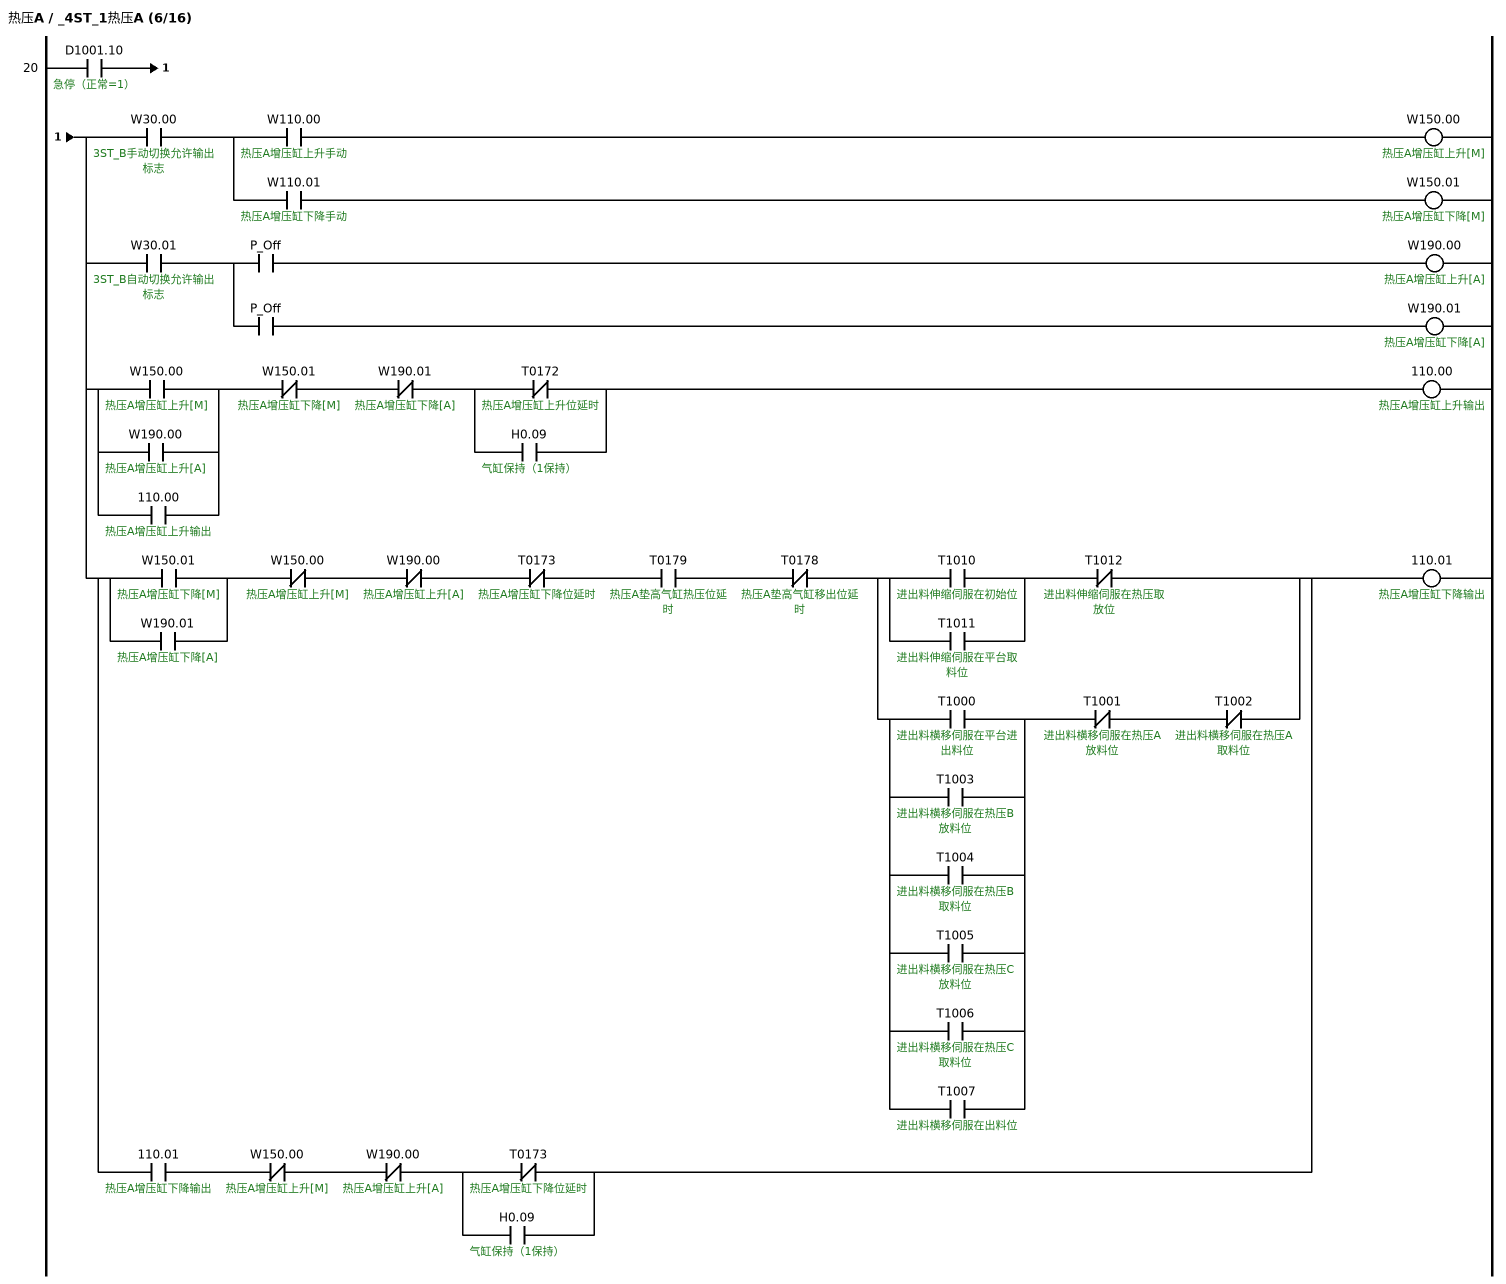
; [picture p144: 热压A / _4ST_1热压A, rungs 20-20]
; rung 20
LD D1001.10  ; 急停（正常=1）
OUT TR0
AND W30.00  ; 3ST_B手动切换允许输出标志
OUT TR1
AND W110.00  ; 热压A增压缸上升手动
OUT W150.00  ; 热压A增压缸上升[M]
LD TR1
AND W110.01  ; 热压A增压缸下降手动
OUT W150.01  ; 热压A增压缸下降[M]
LD TR0
AND W30.01  ; 3ST_B自动切换允许输出标志
OUT TR1
AND P_Off
OUT W190.00  ; 热压A增压缸上升[A]
LD TR1
AND P_Off
OUT W190.01  ; 热压A增压缸下降[A]
LD TR0
LD W150.00  ; 热压A增压缸上升[M]
OR W190.00  ; 热压A增压缸上升[A]
OR 110.00  ; 热压A增压缸上升输出
ANDLD
ANDNOT W150.01  ; 热压A增压缸下降[M]
ANDNOT W190.01  ; 热压A增压缸下降[A]
LDNOT T0172  ; 热压A增压缸上升位延时
OR H0.09  ; 气缸保持（1保持）
ANDLD
OUT 110.00  ; 热压A增压缸上升输出
LD TR0
LD W150.01  ; 热压A增压缸下降[M]
OR W190.01  ; 热压A增压缸下降[A]
ANDNOT W150.00  ; 热压A增压缸上升[M]
ANDNOT W190.00  ; 热压A增压缸上升[A]
ANDNOT T0173  ; 热压A增压缸下降位延时
AND T0179  ; 热压A垫高气缸热压位延时
ANDNOT T0178  ; 热压A垫高气缸移出位延时
LD T1010  ; 进出料伸缩伺服在初始位
OR T1011  ; 进出料伸缩伺服在平台取料位
ANDNOT T1012  ; 进出料伸缩伺服在热压取放位
LD T1000  ; 进出料横移伺服在平台进出料位
OR T1003  ; 进出料横移伺服在热压B放料位
OR T1004  ; 进出料横移伺服在热压B取料位
OR T1005  ; 进出料横移伺服在热压C放料位
OR T1006  ; 进出料横移伺服在热压C取料位
OR T1007  ; 进出料横移伺服在出料位
ANDNOT T1001  ; 进出料横移伺服在热压A放料位
ANDNOT T1002  ; 进出料横移伺服在热压A取料位
ORLD
ANDLD
LD 110.01  ; 热压A增压缸下降输出
ANDNOT W150.00  ; 热压A增压缸上升[M]
ANDNOT W190.00  ; 热压A增压缸上升[A]
LDNOT T0173  ; 热压A增压缸下降位延时
OR H0.09  ; 气缸保持（1保持）
ANDLD
ORLD
ANDLD
OUT 110.01  ; 热压A增压缸下降输出

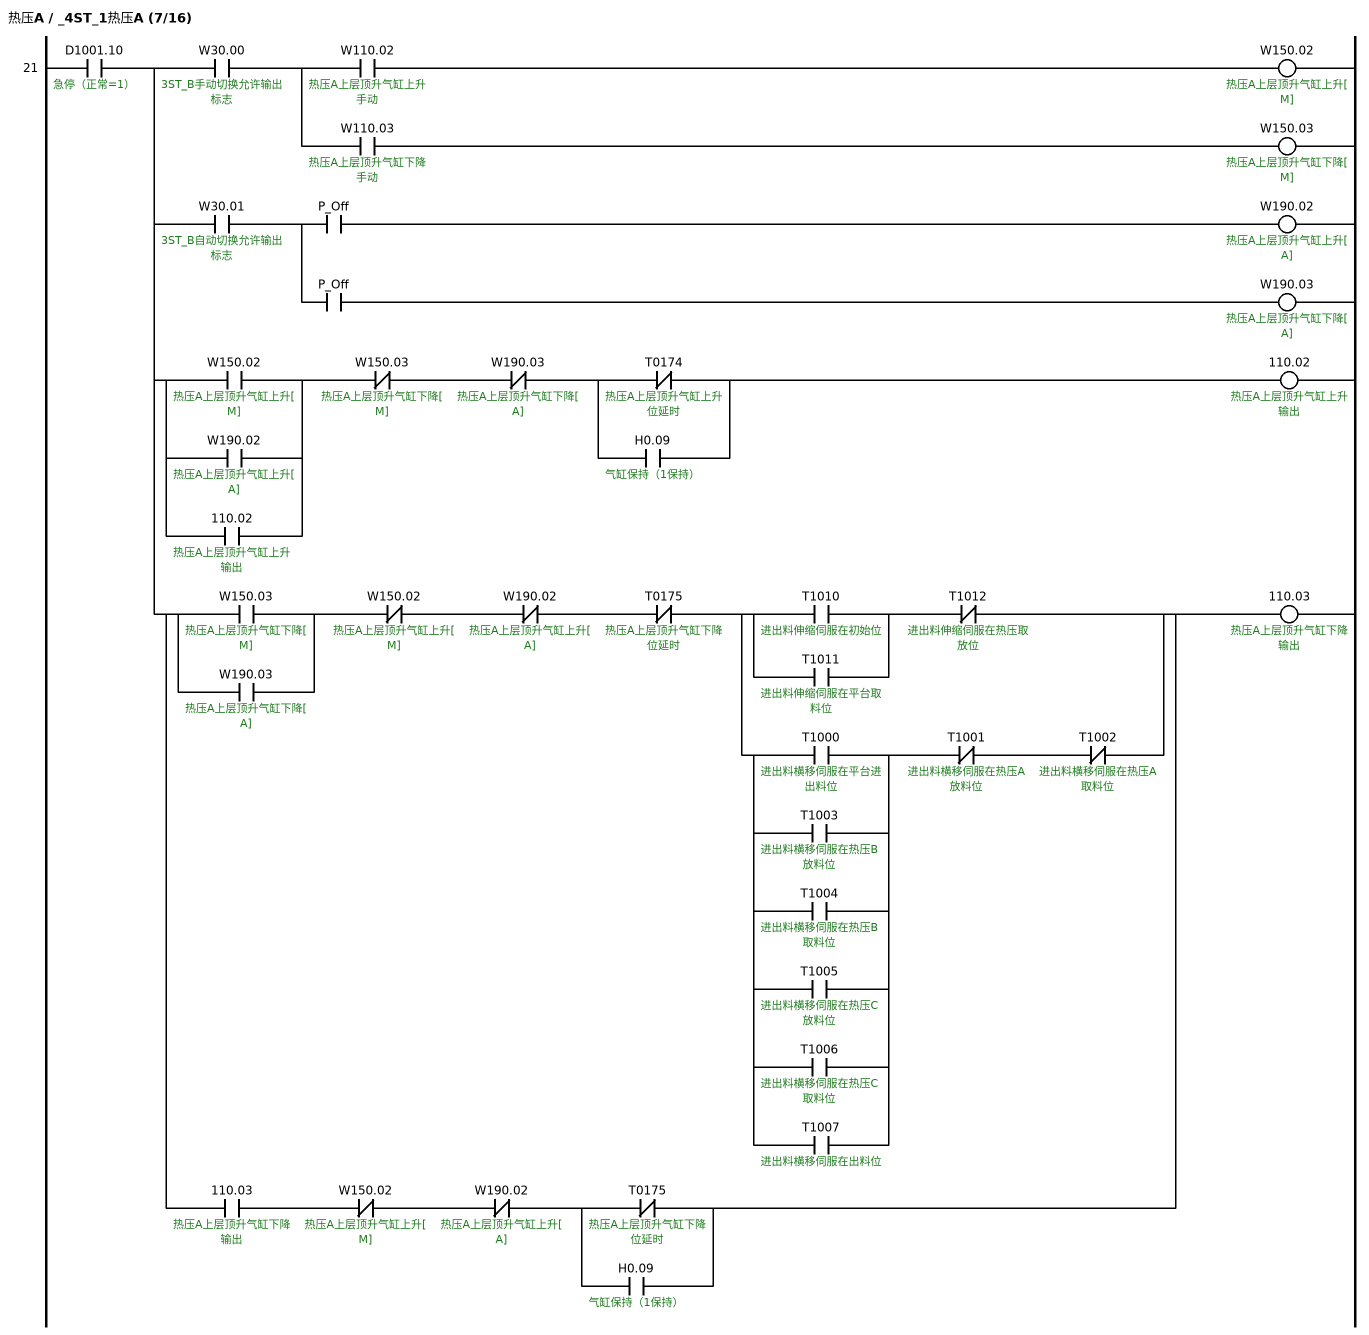
; rung 21
LD D1001.10  ; 急停（正常=1）
OUT TR0
AND W30.00  ; 3ST_B手动切换允许输出标志
OUT TR1
AND W110.02  ; 热压A上层顶升气缸上升手动
OUT W150.02  ; 热压A上层顶升气缸上升[M]
LD TR1
AND W110.03  ; 热压A上层顶升气缸下降手动
OUT W150.03  ; 热压A上层顶升气缸下降[M]
LD TR0
AND W30.01  ; 3ST_B自动切换允许输出标志
OUT TR1
AND P_Off
OUT W190.02  ; 热压A上层顶升气缸上升[A]
LD TR1
AND P_Off
OUT W190.03  ; 热压A上层顶升气缸下降[A]
LD TR0
LD W150.02  ; 热压A上层顶升气缸上升[M]
OR W190.02  ; 热压A上层顶升气缸上升[A]
OR 110.02  ; 热压A上层顶升气缸上升输出
ANDLD
ANDNOT W150.03  ; 热压A上层顶升气缸下降[M]
ANDNOT W190.03  ; 热压A上层顶升气缸下降[A]
LDNOT T0174  ; 热压A上层顶升气缸上升位延时
OR H0.09  ; 气缸保持（1保持）
ANDLD
OUT 110.02  ; 热压A上层顶升气缸上升输出
LD TR0
LD W150.03  ; 热压A上层顶升气缸下降[M]
OR W190.03  ; 热压A上层顶升气缸下降[A]
ANDNOT W150.02  ; 热压A上层顶升气缸上升[M]
ANDNOT W190.02  ; 热压A上层顶升气缸上升[A]
ANDNOT T0175  ; 热压A上层顶升气缸下降位延时
LD T1010  ; 进出料伸缩伺服在初始位
OR T1011  ; 进出料伸缩伺服在平台取料位
ANDNOT T1012  ; 进出料伸缩伺服在热压取放位
LD T1000  ; 进出料横移伺服在平台进出料位
OR T1003  ; 进出料横移伺服在热压B放料位
OR T1004  ; 进出料横移伺服在热压B取料位
OR T1005  ; 进出料横移伺服在热压C放料位
OR T1006  ; 进出料横移伺服在热压C取料位
OR T1007  ; 进出料横移伺服在出料位
ANDNOT T1001  ; 进出料横移伺服在热压A放料位
ANDNOT T1002  ; 进出料横移伺服在热压A取料位
ORLD
ANDLD
LD 110.03  ; 热压A上层顶升气缸下降输出
ANDNOT W150.02  ; 热压A上层顶升气缸上升[M]
ANDNOT W190.02  ; 热压A上层顶升气缸上升[A]
LDNOT T0175  ; 热压A上层顶升气缸下降位延时
OR H0.09  ; 气缸保持（1保持）
ANDLD
ORLD
ANDLD
OUT 110.03  ; 热压A上层顶升气缸下降输出

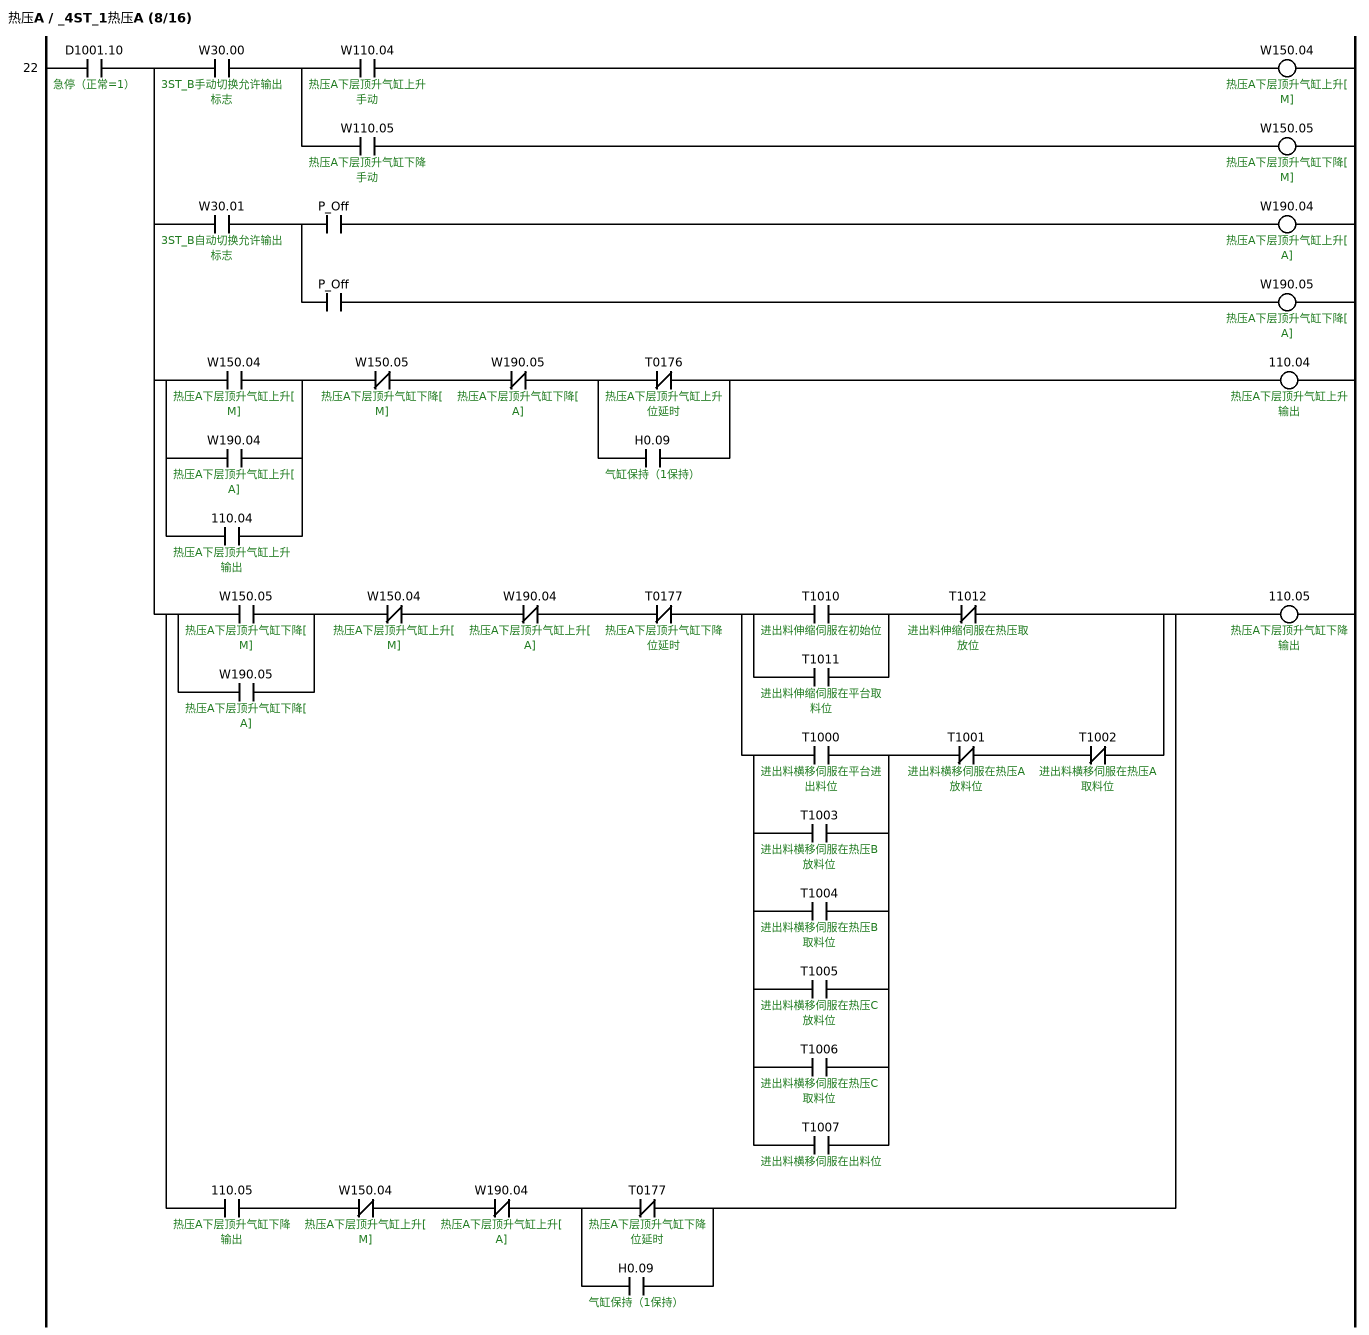
; rung 22
LD D1001.10  ; 急停（正常=1）
OUT TR0
AND W30.00  ; 3ST_B手动切换允许输出标志
OUT TR1
AND W110.04  ; 热压A下层顶升气缸上升手动
OUT W150.04  ; 热压A下层顶升气缸上升[M]
LD TR1
AND W110.05  ; 热压A下层顶升气缸下降手动
OUT W150.05  ; 热压A下层顶升气缸下降[M]
LD TR0
AND W30.01  ; 3ST_B自动切换允许输出标志
OUT TR1
AND P_Off
OUT W190.04  ; 热压A下层顶升气缸上升[A]
LD TR1
AND P_Off
OUT W190.05  ; 热压A下层顶升气缸下降[A]
LD TR0
LD W150.04  ; 热压A下层顶升气缸上升[M]
OR W190.04  ; 热压A下层顶升气缸上升[A]
OR 110.04  ; 热压A下层顶升气缸上升输出
ANDLD
ANDNOT W150.05  ; 热压A下层顶升气缸下降[M]
ANDNOT W190.05  ; 热压A下层顶升气缸下降[A]
LDNOT T0176  ; 热压A下层顶升气缸上升位延时
OR H0.09  ; 气缸保持（1保持）
ANDLD
OUT 110.04  ; 热压A下层顶升气缸上升输出
LD TR0
LD W150.05  ; 热压A下层顶升气缸下降[M]
OR W190.05  ; 热压A下层顶升气缸下降[A]
ANDNOT W150.04  ; 热压A下层顶升气缸上升[M]
ANDNOT W190.04  ; 热压A下层顶升气缸上升[A]
ANDNOT T0177  ; 热压A下层顶升气缸下降位延时
LD T1010  ; 进出料伸缩伺服在初始位
OR T1011  ; 进出料伸缩伺服在平台取料位
ANDNOT T1012  ; 进出料伸缩伺服在热压取放位
LD T1000  ; 进出料横移伺服在平台进出料位
OR T1003  ; 进出料横移伺服在热压B放料位
OR T1004  ; 进出料横移伺服在热压B取料位
OR T1005  ; 进出料横移伺服在热压C放料位
OR T1006  ; 进出料横移伺服在热压C取料位
OR T1007  ; 进出料横移伺服在出料位
ANDNOT T1001  ; 进出料横移伺服在热压A放料位
ANDNOT T1002  ; 进出料横移伺服在热压A取料位
ORLD
ANDLD
LD 110.05  ; 热压A下层顶升气缸下降输出
ANDNOT W150.04  ; 热压A下层顶升气缸上升[M]
ANDNOT W190.04  ; 热压A下层顶升气缸上升[A]
LDNOT T0177  ; 热压A下层顶升气缸下降位延时
OR H0.09  ; 气缸保持（1保持）
ANDLD
ORLD
ANDLD
OUT 110.05  ; 热压A下层顶升气缸下降输出

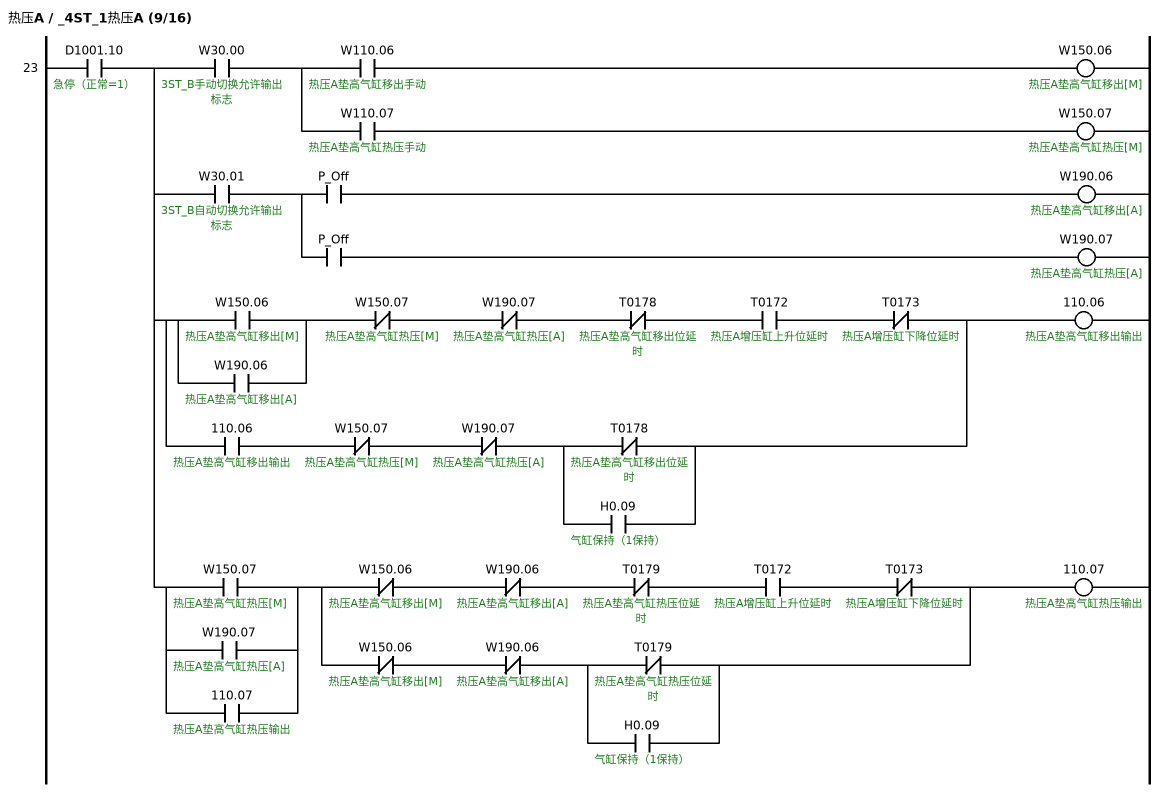
; rung 23
LD D1001.10  ; 急停（正常=1）
OUT TR0
AND W30.00  ; 3ST_B手动切换允许输出标志
OUT TR1
AND W110.06  ; 热压A垫高气缸移出手动
OUT W150.06  ; 热压A垫高气缸移出[M]
LD TR1
AND W110.07  ; 热压A垫高气缸热压手动
OUT W150.07  ; 热压A垫高气缸热压[M]
LD TR0
AND W30.01  ; 3ST_B自动切换允许输出标志
OUT TR1
AND P_Off
OUT W190.06  ; 热压A垫高气缸移出[A]
LD TR1
AND P_Off
OUT W190.07  ; 热压A垫高气缸热压[A]
LD TR0
LD W150.06  ; 热压A垫高气缸移出[M]
OR W190.06  ; 热压A垫高气缸移出[A]
ANDNOT W150.07  ; 热压A垫高气缸热压[M]
ANDNOT W190.07  ; 热压A垫高气缸热压[A]
ANDNOT T0178  ; 热压A垫高气缸移出位延时
AND T0172  ; 热压A增压缸上升位延时
ANDNOT T0173  ; 热压A增压缸下降位延时
LD 110.06  ; 热压A垫高气缸移出输出
ANDNOT W150.07  ; 热压A垫高气缸热压[M]
ANDNOT W190.07  ; 热压A垫高气缸热压[A]
LDNOT T0178  ; 热压A垫高气缸移出位延时
OR H0.09  ; 气缸保持（1保持）
ANDLD
ORLD
ANDLD
OUT 110.06  ; 热压A垫高气缸移出输出
LD TR0
LD W150.07  ; 热压A垫高气缸热压[M]
OR W190.07  ; 热压A垫高气缸热压[A]
OR 110.07  ; 热压A垫高气缸热压输出
ANDLD
LDNOT W150.06  ; 热压A垫高气缸移出[M]
ANDNOT W190.06  ; 热压A垫高气缸移出[A]
ANDNOT T0179  ; 热压A垫高气缸热压位延时
AND T0172  ; 热压A增压缸上升位延时
ANDNOT T0173  ; 热压A增压缸下降位延时
LDNOT W150.06  ; 热压A垫高气缸移出[M]
ANDNOT W190.06  ; 热压A垫高气缸移出[A]
LDNOT T0179  ; 热压A垫高气缸热压位延时
OR H0.09  ; 气缸保持（1保持）
ANDLD
ORLD
ANDLD
OUT 110.07  ; 热压A垫高气缸热压输出

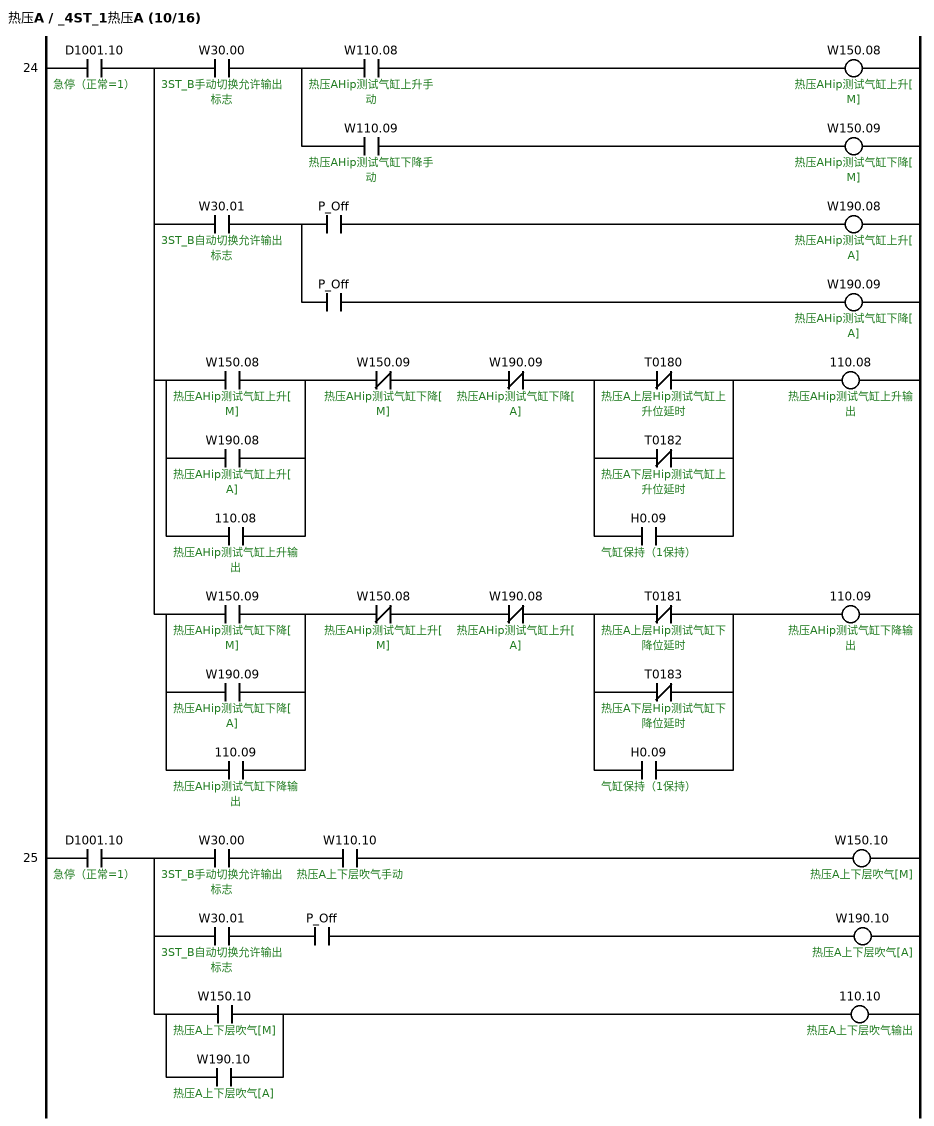
; rung 24
LD D1001.10  ; 急停（正常=1）
OUT TR0
AND W30.00  ; 3ST_B手动切换允许输出标志
OUT TR1
AND W110.08  ; 热压AHip测试气缸上升手动
OUT W150.08  ; 热压AHip测试气缸上升[M]
LD TR1
AND W110.09  ; 热压AHip测试气缸下降手动
OUT W150.09  ; 热压AHip测试气缸下降[M]
LD TR0
AND W30.01  ; 3ST_B自动切换允许输出标志
OUT TR1
AND P_Off
OUT W190.08  ; 热压AHip测试气缸上升[A]
LD TR1
AND P_Off
OUT W190.09  ; 热压AHip测试气缸下降[A]
LD TR0
LD W150.08  ; 热压AHip测试气缸上升[M]
OR W190.08  ; 热压AHip测试气缸上升[A]
OR 110.08  ; 热压AHip测试气缸上升输出
ANDLD
ANDNOT W150.09  ; 热压AHip测试气缸下降[M]
ANDNOT W190.09  ; 热压AHip测试气缸下降[A]
LDNOT T0180  ; 热压A上层Hip测试气缸上升位延时
ORNOT T0182  ; 热压A下层Hip测试气缸上升位延时
OR H0.09  ; 气缸保持（1保持）
ANDLD
OUT 110.08  ; 热压AHip测试气缸上升输出
LD TR0
LD W150.09  ; 热压AHip测试气缸下降[M]
OR W190.09  ; 热压AHip测试气缸下降[A]
OR 110.09  ; 热压AHip测试气缸下降输出
ANDLD
ANDNOT W150.08  ; 热压AHip测试气缸上升[M]
ANDNOT W190.08  ; 热压AHip测试气缸上升[A]
LDNOT T0181  ; 热压A上层Hip测试气缸下降位延时
ORNOT T0183  ; 热压A下层Hip测试气缸下降位延时
OR H0.09  ; 气缸保持（1保持）
ANDLD
OUT 110.09  ; 热压AHip测试气缸下降输出
; rung 25
LD D1001.10  ; 急停（正常=1）
OUT TR0
AND W30.00  ; 3ST_B手动切换允许输出标志
AND W110.10  ; 热压A上下层吹气手动
OUT W150.10  ; 热压A上下层吹气[M]
LD TR0
AND W30.01  ; 3ST_B自动切换允许输出标志
AND P_Off
OUT W190.10  ; 热压A上下层吹气[A]
LD TR0
LD W150.10  ; 热压A上下层吹气[M]
OR W190.10  ; 热压A上下层吹气[A]
ANDLD
OUT 110.10  ; 热压A上下层吹气输出

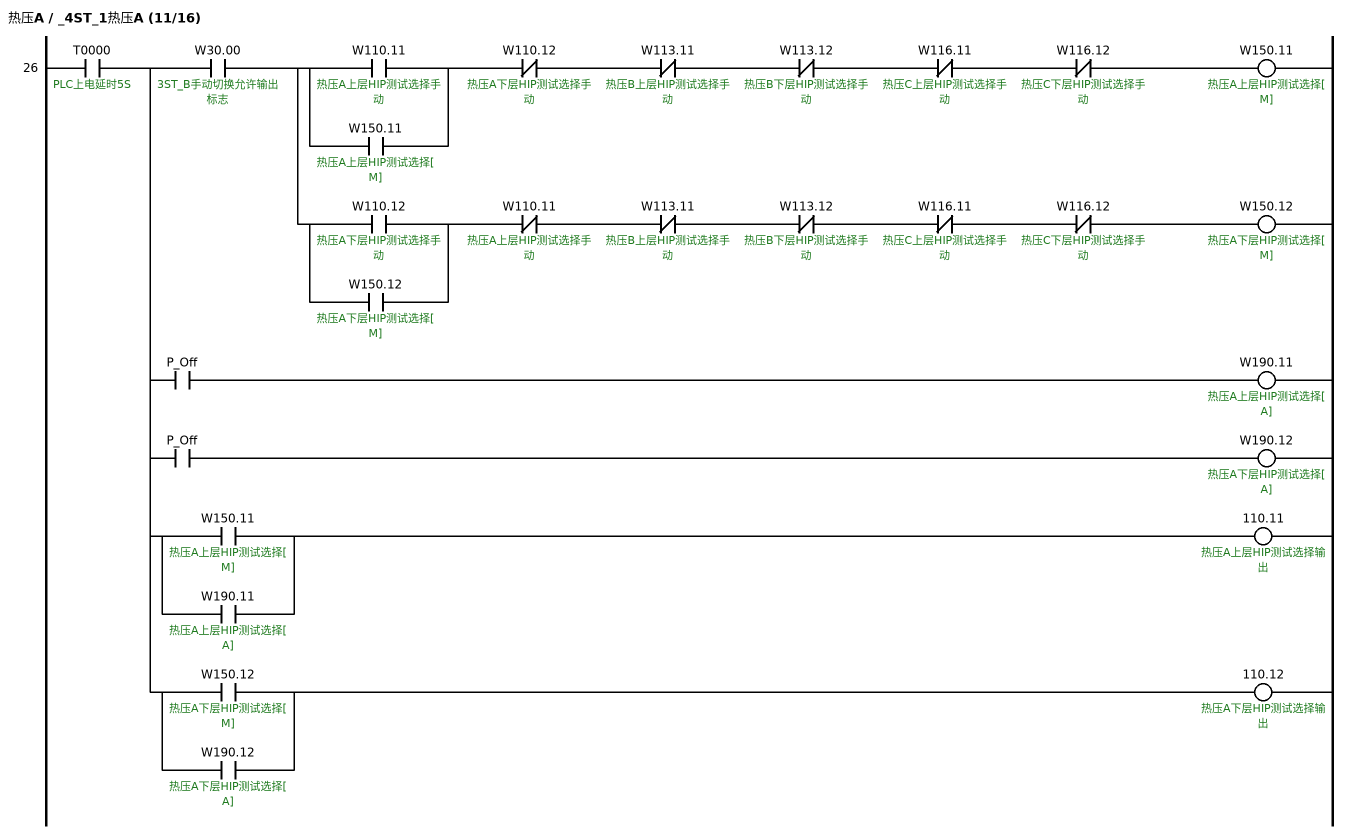
; rung 26
LD T0000  ; PLC上电延时5S
OUT TR0
AND W30.00  ; 3ST_B手动切换允许输出标志
OUT TR1
LD W110.11  ; 热压A上层HIP测试选择手动
OR W150.11  ; 热压A上层HIP测试选择[M]
ANDLD
ANDNOT W110.12  ; 热压A下层HIP测试选择手动
ANDNOT W113.11  ; 热压B上层HIP测试选择手动
ANDNOT W113.12  ; 热压B下层HIP测试选择手动
ANDNOT W116.11  ; 热压C上层HIP测试选择手动
ANDNOT W116.12  ; 热压C下层HIP测试选择手动
OUT W150.11  ; 热压A上层HIP测试选择[M]
LD TR1
LD W110.12  ; 热压A下层HIP测试选择手动
OR W150.12  ; 热压A下层HIP测试选择[M]
ANDLD
ANDNOT W110.11  ; 热压A上层HIP测试选择手动
ANDNOT W113.11  ; 热压B上层HIP测试选择手动
ANDNOT W113.12  ; 热压B下层HIP测试选择手动
ANDNOT W116.11  ; 热压C上层HIP测试选择手动
ANDNOT W116.12  ; 热压C下层HIP测试选择手动
OUT W150.12  ; 热压A下层HIP测试选择[M]
LD TR0
AND P_Off
OUT W190.11  ; 热压A上层HIP测试选择[A]
LD TR0
AND P_Off
OUT W190.12  ; 热压A下层HIP测试选择[A]
LD TR0
LD W150.11  ; 热压A上层HIP测试选择[M]
OR W190.11  ; 热压A上层HIP测试选择[A]
ANDLD
OUT 110.11  ; 热压A上层HIP测试选择输出
LD TR0
LD W150.12  ; 热压A下层HIP测试选择[M]
OR W190.12  ; 热压A下层HIP测试选择[A]
ANDLD
OUT 110.12  ; 热压A下层HIP测试选择输出

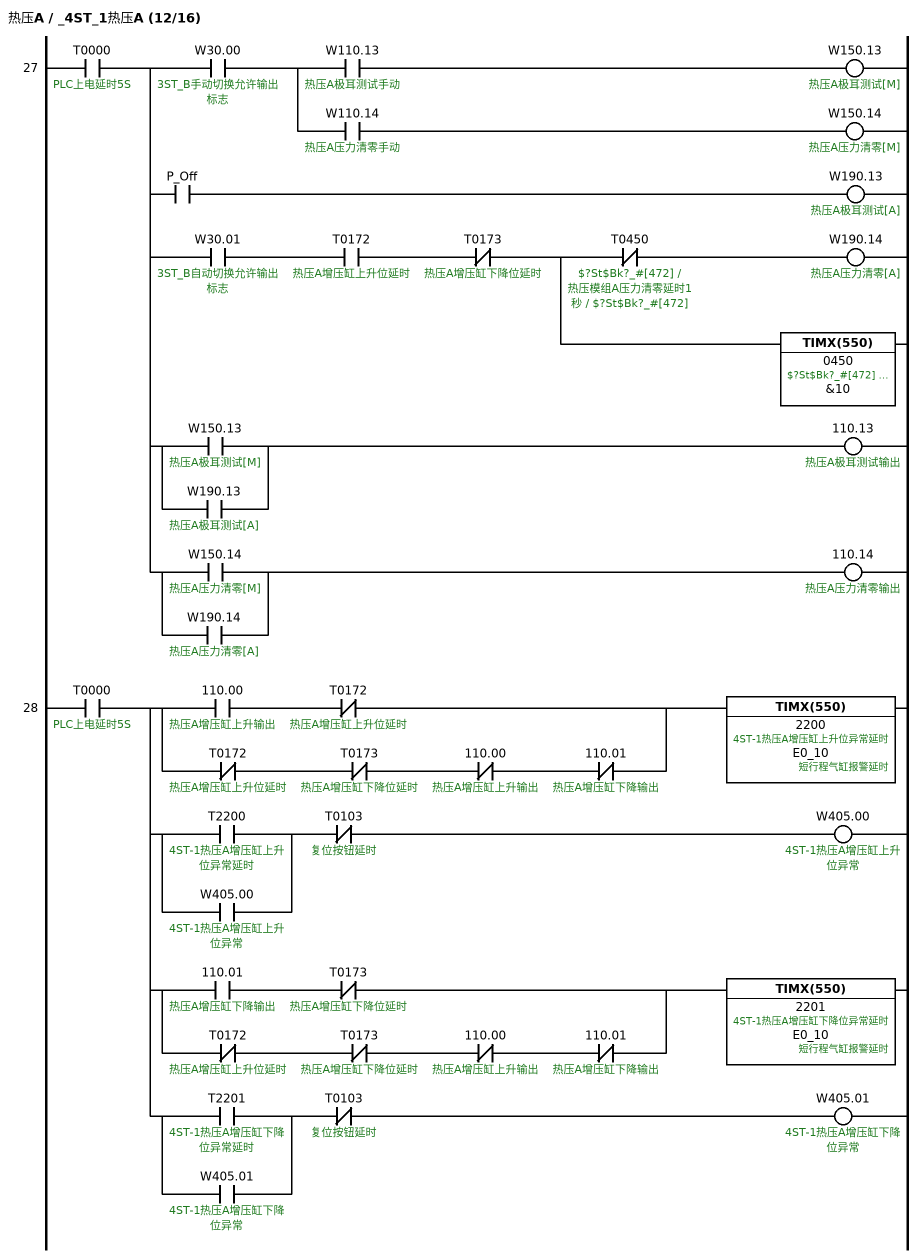
; rung 27
LD T0000  ; PLC上电延时5S
OUT TR0
AND W30.00  ; 3ST_B手动切换允许输出标志
OUT TR1
AND W110.13  ; 热压A极耳测试手动
OUT W150.13  ; 热压A极耳测试[M]
LD TR1
AND W110.14  ; 热压A压力清零手动
OUT W150.14  ; 热压A压力清零[M]
LD TR0
AND P_Off
OUT W190.13  ; 热压A极耳测试[A]
LD TR0
AND W30.01  ; 3ST_B自动切换允许输出标志
AND T0172  ; 热压A增压缸上升位延时
ANDNOT T0173  ; 热压A增压缸下降位延时
OUT TR1
ANDNOT T0450  ; $?St$Bk?_#[472] / 热压模组A压力清零延时1秒 / $?St$Bk?_#[472]
OUT W190.14  ; 热压A压力清零[A]
LD TR1
TIMX(550) 0450 &10  ; $?St$Bk?_#[472] / 热压模组A压力清零延时1秒 / $?St$Bk?_#[472]
LD TR0
LD W150.13  ; 热压A极耳测试[M]
OR W190.13  ; 热压A极耳测试[A]
ANDLD
OUT 110.13  ; 热压A极耳测试输出
LD TR0
LD W150.14  ; 热压A压力清零[M]
OR W190.14  ; 热压A压力清零[A]
ANDLD
OUT 110.14  ; 热压A压力清零输出
; rung 28
LD T0000  ; PLC上电延时5S
OUT TR0
LD 110.00  ; 热压A增压缸上升输出
ANDNOT T0172  ; 热压A增压缸上升位延时
LDNOT T0172  ; 热压A增压缸上升位延时
ANDNOT T0173  ; 热压A增压缸下降位延时
ANDNOT 110.00  ; 热压A增压缸上升输出
ANDNOT 110.01  ; 热压A增压缸下降输出
ORLD
ANDLD
TIMX(550) 2200 E0_10  ; 短行程气缸报警延时, 4ST-1热压A增压缸上升位异常延时
LD TR0
LD T2200  ; 4ST-1热压A增压缸上升位异常延时
OR W405.00  ; 4ST-1热压A增压缸上升位异常
ANDLD
ANDNOT T0103  ; 复位按钮延时
OUT W405.00  ; 4ST-1热压A增压缸上升位异常
LD TR0
LD 110.01  ; 热压A增压缸下降输出
ANDNOT T0173  ; 热压A增压缸下降位延时
LDNOT T0172  ; 热压A增压缸上升位延时
ANDNOT T0173  ; 热压A增压缸下降位延时
ANDNOT 110.00  ; 热压A增压缸上升输出
ANDNOT 110.01  ; 热压A增压缸下降输出
ORLD
ANDLD
TIMX(550) 2201 E0_10  ; 短行程气缸报警延时, 4ST-1热压A增压缸下降位异常延时
LD TR0
LD T2201  ; 4ST-1热压A增压缸下降位异常延时
OR W405.01  ; 4ST-1热压A增压缸下降位异常
ANDLD
ANDNOT T0103  ; 复位按钮延时
OUT W405.01  ; 4ST-1热压A增压缸下降位异常

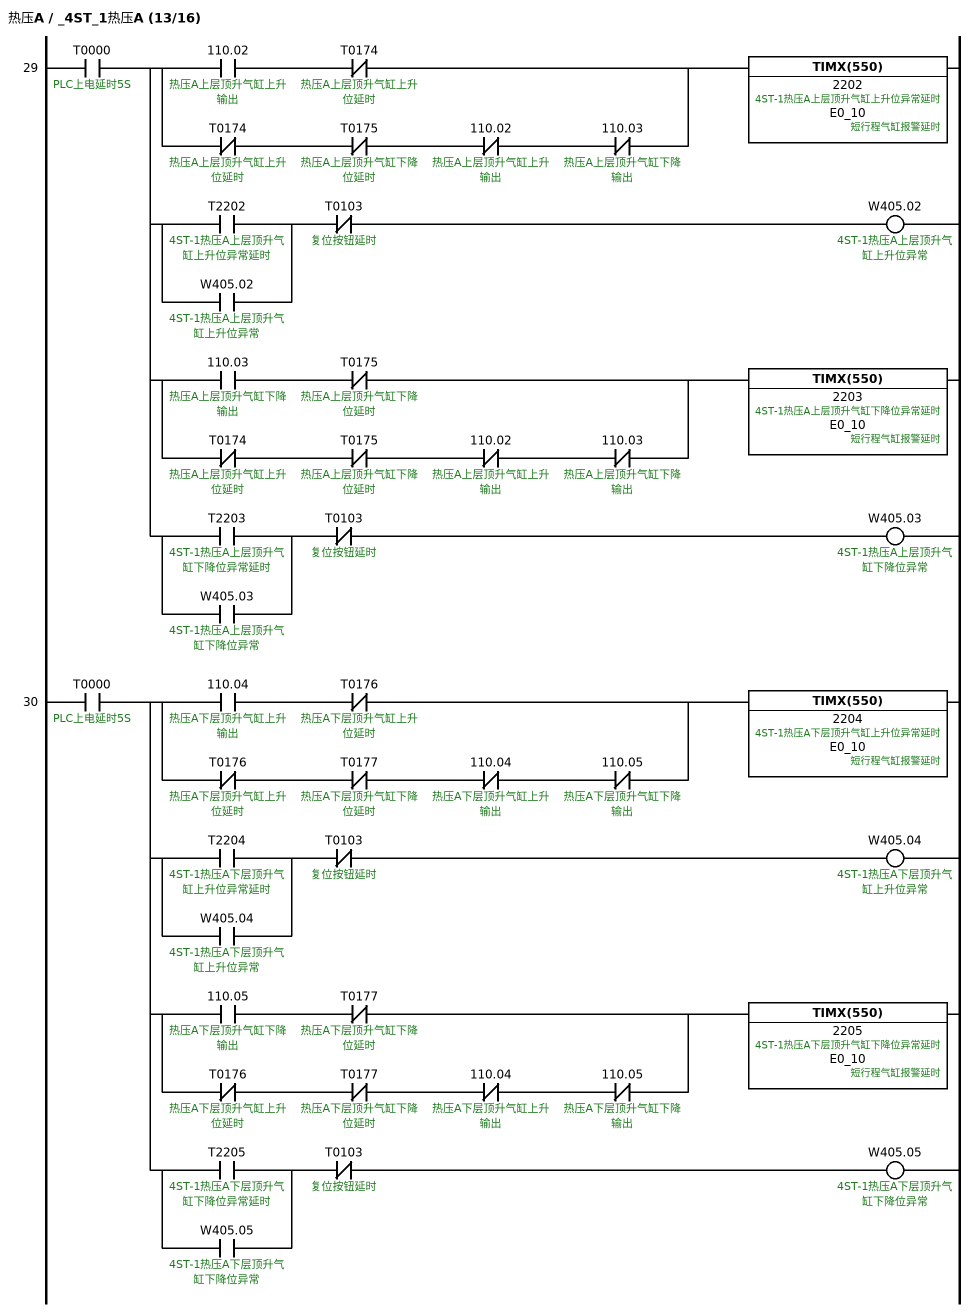
; rung 29
LD T0000  ; PLC上电延时5S
OUT TR0
LD 110.02  ; 热压A上层顶升气缸上升输出
ANDNOT T0174  ; 热压A上层顶升气缸上升位延时
LDNOT T0174  ; 热压A上层顶升气缸上升位延时
ANDNOT T0175  ; 热压A上层顶升气缸下降位延时
ANDNOT 110.02  ; 热压A上层顶升气缸上升输出
ANDNOT 110.03  ; 热压A上层顶升气缸下降输出
ORLD
ANDLD
TIMX(550) 2202 E0_10  ; 短行程气缸报警延时, 4ST-1热压A上层顶升气缸上升位异常延时
LD TR0
LD T2202  ; 4ST-1热压A上层顶升气缸上升位异常延时
OR W405.02  ; 4ST-1热压A上层顶升气缸上升位异常
ANDLD
ANDNOT T0103  ; 复位按钮延时
OUT W405.02  ; 4ST-1热压A上层顶升气缸上升位异常
LD TR0
LD 110.03  ; 热压A上层顶升气缸下降输出
ANDNOT T0175  ; 热压A上层顶升气缸下降位延时
LDNOT T0174  ; 热压A上层顶升气缸上升位延时
ANDNOT T0175  ; 热压A上层顶升气缸下降位延时
ANDNOT 110.02  ; 热压A上层顶升气缸上升输出
ANDNOT 110.03  ; 热压A上层顶升气缸下降输出
ORLD
ANDLD
TIMX(550) 2203 E0_10  ; 短行程气缸报警延时, 4ST-1热压A上层顶升气缸下降位异常延时
LD TR0
LD T2203  ; 4ST-1热压A上层顶升气缸下降位异常延时
OR W405.03  ; 4ST-1热压A上层顶升气缸下降位异常
ANDLD
ANDNOT T0103  ; 复位按钮延时
OUT W405.03  ; 4ST-1热压A上层顶升气缸下降位异常
; rung 30
LD T0000  ; PLC上电延时5S
OUT TR0
LD 110.04  ; 热压A下层顶升气缸上升输出
ANDNOT T0176  ; 热压A下层顶升气缸上升位延时
LDNOT T0176  ; 热压A下层顶升气缸上升位延时
ANDNOT T0177  ; 热压A下层顶升气缸下降位延时
ANDNOT 110.04  ; 热压A下层顶升气缸上升输出
ANDNOT 110.05  ; 热压A下层顶升气缸下降输出
ORLD
ANDLD
TIMX(550) 2204 E0_10  ; 短行程气缸报警延时, 4ST-1热压A下层顶升气缸上升位异常延时
LD TR0
LD T2204  ; 4ST-1热压A下层顶升气缸上升位异常延时
OR W405.04  ; 4ST-1热压A下层顶升气缸上升位异常
ANDLD
ANDNOT T0103  ; 复位按钮延时
OUT W405.04  ; 4ST-1热压A下层顶升气缸上升位异常
LD TR0
LD 110.05  ; 热压A下层顶升气缸下降输出
ANDNOT T0177  ; 热压A下层顶升气缸下降位延时
LDNOT T0176  ; 热压A下层顶升气缸上升位延时
ANDNOT T0177  ; 热压A下层顶升气缸下降位延时
ANDNOT 110.04  ; 热压A下层顶升气缸上升输出
ANDNOT 110.05  ; 热压A下层顶升气缸下降输出
ORLD
ANDLD
TIMX(550) 2205 E0_10  ; 短行程气缸报警延时, 4ST-1热压A下层顶升气缸下降位异常延时
LD TR0
LD T2205  ; 4ST-1热压A下层顶升气缸下降位异常延时
OR W405.05  ; 4ST-1热压A下层顶升气缸下降位异常
ANDLD
ANDNOT T0103  ; 复位按钮延时
OUT W405.05  ; 4ST-1热压A下层顶升气缸下降位异常

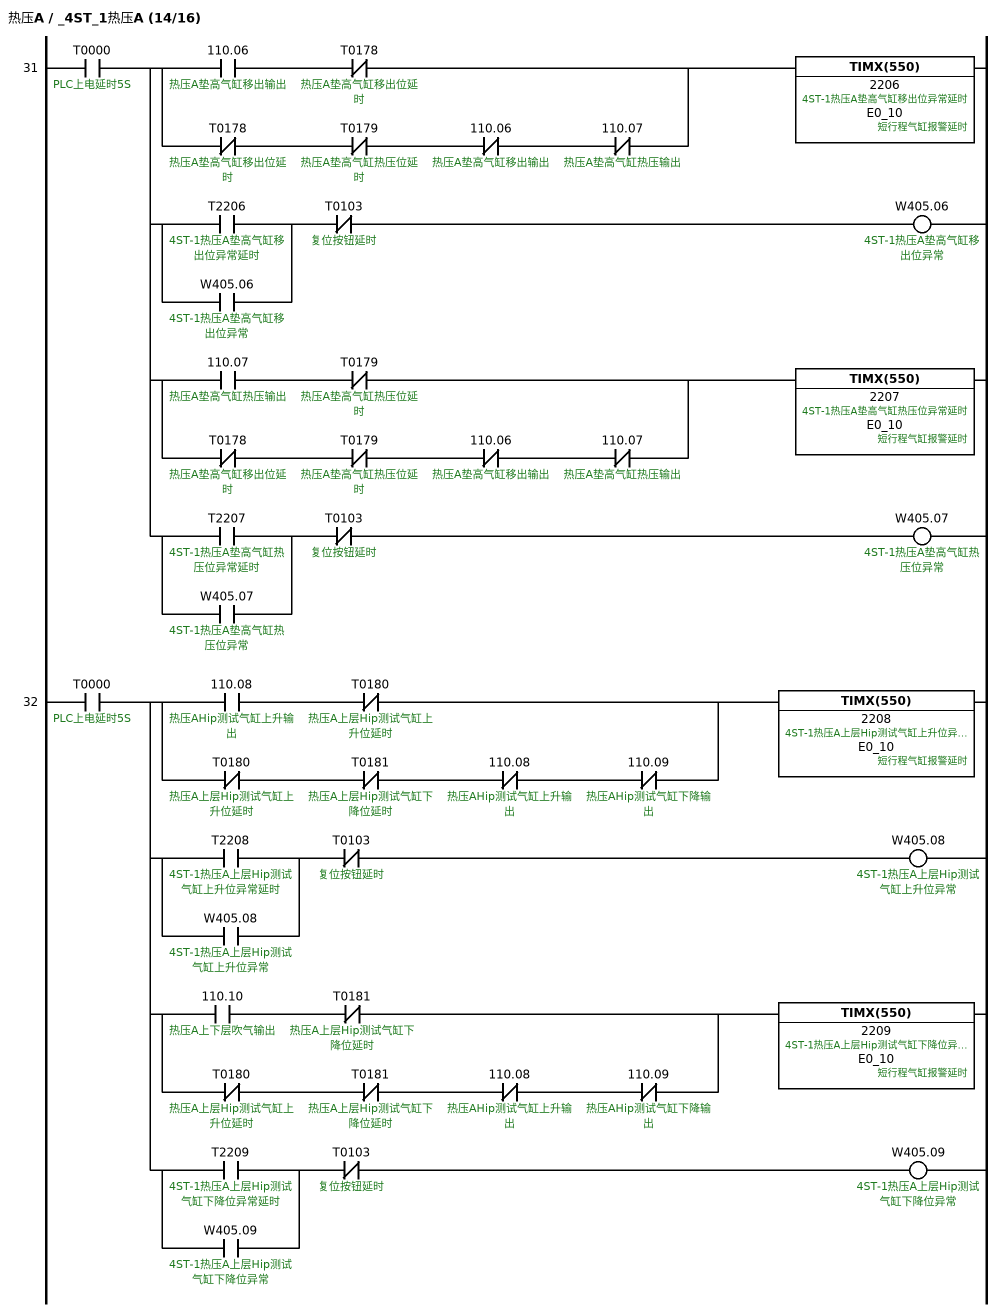
; rung 31
LD T0000  ; PLC上电延时5S
OUT TR0
LD 110.06  ; 热压A垫高气缸移出输出
ANDNOT T0178  ; 热压A垫高气缸移出位延时
LDNOT T0178  ; 热压A垫高气缸移出位延时
ANDNOT T0179  ; 热压A垫高气缸热压位延时
ANDNOT 110.06  ; 热压A垫高气缸移出输出
ANDNOT 110.07  ; 热压A垫高气缸热压输出
ORLD
ANDLD
TIMX(550) 2206 E0_10  ; 短行程气缸报警延时, 4ST-1热压A垫高气缸移出位异常延时
LD TR0
LD T2206  ; 4ST-1热压A垫高气缸移出位异常延时
OR W405.06  ; 4ST-1热压A垫高气缸移出位异常
ANDLD
ANDNOT T0103  ; 复位按钮延时
OUT W405.06  ; 4ST-1热压A垫高气缸移出位异常
LD TR0
LD 110.07  ; 热压A垫高气缸热压输出
ANDNOT T0179  ; 热压A垫高气缸热压位延时
LDNOT T0178  ; 热压A垫高气缸移出位延时
ANDNOT T0179  ; 热压A垫高气缸热压位延时
ANDNOT 110.06  ; 热压A垫高气缸移出输出
ANDNOT 110.07  ; 热压A垫高气缸热压输出
ORLD
ANDLD
TIMX(550) 2207 E0_10  ; 短行程气缸报警延时, 4ST-1热压A垫高气缸热压位异常延时
LD TR0
LD T2207  ; 4ST-1热压A垫高气缸热压位异常延时
OR W405.07  ; 4ST-1热压A垫高气缸热压位异常
ANDLD
ANDNOT T0103  ; 复位按钮延时
OUT W405.07  ; 4ST-1热压A垫高气缸热压位异常
; rung 32
LD T0000  ; PLC上电延时5S
OUT TR0
LD 110.08  ; 热压AHip测试气缸上升输出
ANDNOT T0180  ; 热压A上层Hip测试气缸上升位延时
LDNOT T0180  ; 热压A上层Hip测试气缸上升位延时
ANDNOT T0181  ; 热压A上层Hip测试气缸下降位延时
ANDNOT 110.08  ; 热压AHip测试气缸上升输出
ANDNOT 110.09  ; 热压AHip测试气缸下降输出
ORLD
ANDLD
TIMX(550) 2208 E0_10  ; 短行程气缸报警延时, 4ST-1热压A上层Hip测试气缸上升位异常延时
LD TR0
LD T2208  ; 4ST-1热压A上层Hip测试气缸上升位异常延时
OR W405.08  ; 4ST-1热压A上层Hip测试气缸上升位异常
ANDLD
ANDNOT T0103  ; 复位按钮延时
OUT W405.08  ; 4ST-1热压A上层Hip测试气缸上升位异常
LD TR0
LD 110.10  ; 热压A上下层吹气输出
ANDNOT T0181  ; 热压A上层Hip测试气缸下降位延时
LDNOT T0180  ; 热压A上层Hip测试气缸上升位延时
ANDNOT T0181  ; 热压A上层Hip测试气缸下降位延时
ANDNOT 110.08  ; 热压AHip测试气缸上升输出
ANDNOT 110.09  ; 热压AHip测试气缸下降输出
ORLD
ANDLD
TIMX(550) 2209 E0_10  ; 短行程气缸报警延时, 4ST-1热压A上层Hip测试气缸下降位异常延时
LD TR0
LD T2209  ; 4ST-1热压A上层Hip测试气缸下降位异常延时
OR W405.09  ; 4ST-1热压A上层Hip测试气缸下降位异常
ANDLD
ANDNOT T0103  ; 复位按钮延时
OUT W405.09  ; 4ST-1热压A上层Hip测试气缸下降位异常

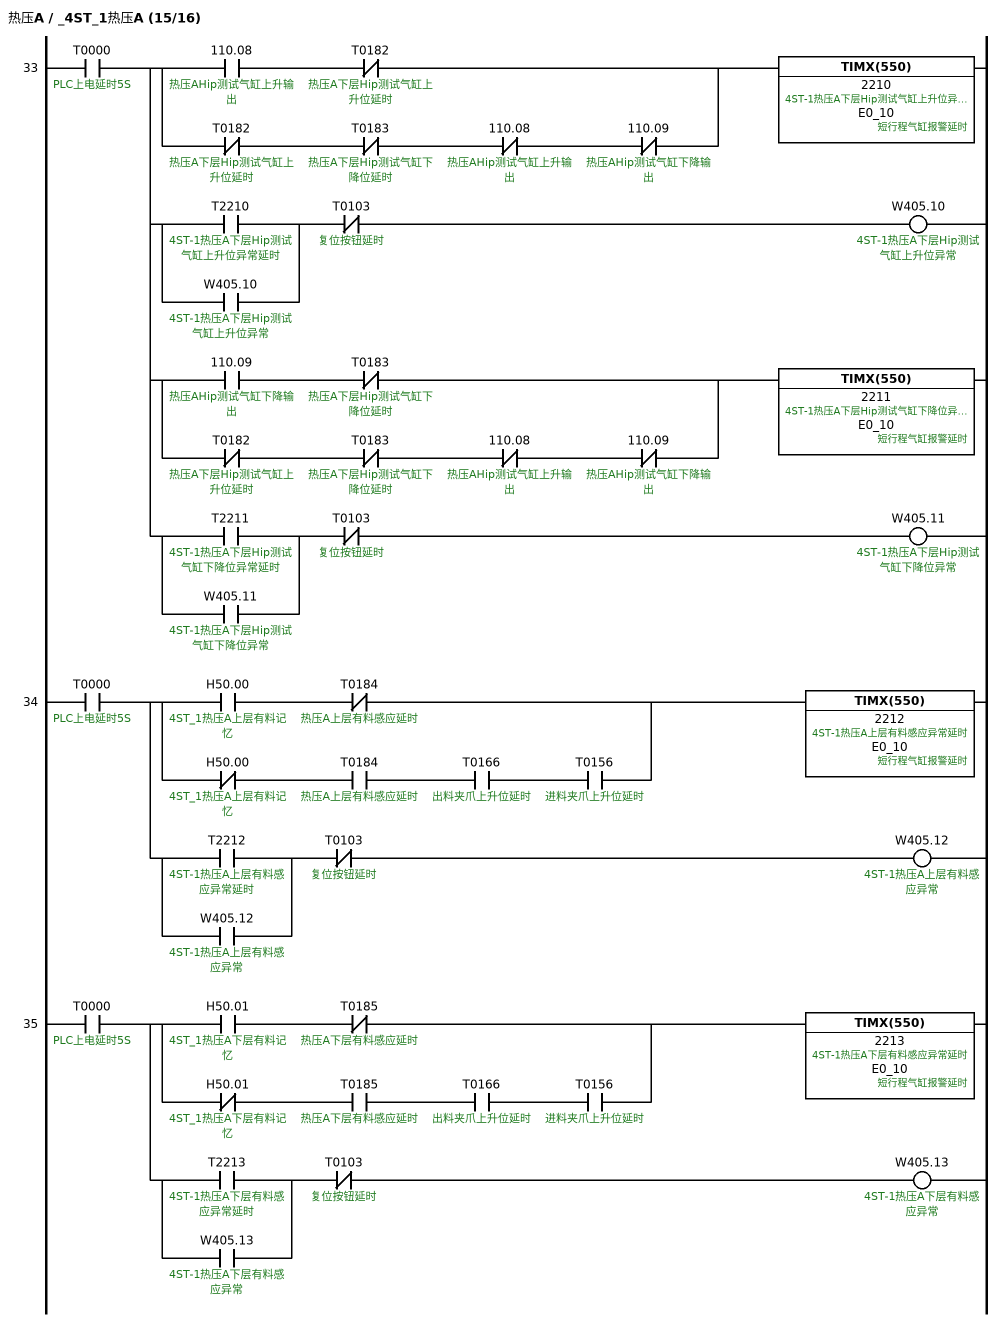
; rung 33
LD T0000  ; PLC上电延时5S
OUT TR0
LD 110.08  ; 热压AHip测试气缸上升输出
ANDNOT T0182  ; 热压A下层Hip测试气缸上升位延时
LDNOT T0182  ; 热压A下层Hip测试气缸上升位延时
ANDNOT T0183  ; 热压A下层Hip测试气缸下降位延时
ANDNOT 110.08  ; 热压AHip测试气缸上升输出
ANDNOT 110.09  ; 热压AHip测试气缸下降输出
ORLD
ANDLD
TIMX(550) 2210 E0_10  ; 短行程气缸报警延时, 4ST-1热压A下层Hip测试气缸上升位异常延时
LD TR0
LD T2210  ; 4ST-1热压A下层Hip测试气缸上升位异常延时
OR W405.10  ; 4ST-1热压A下层Hip测试气缸上升位异常
ANDLD
ANDNOT T0103  ; 复位按钮延时
OUT W405.10  ; 4ST-1热压A下层Hip测试气缸上升位异常
LD TR0
LD 110.09  ; 热压AHip测试气缸下降输出
ANDNOT T0183  ; 热压A下层Hip测试气缸下降位延时
LDNOT T0182  ; 热压A下层Hip测试气缸上升位延时
ANDNOT T0183  ; 热压A下层Hip测试气缸下降位延时
ANDNOT 110.08  ; 热压AHip测试气缸上升输出
ANDNOT 110.09  ; 热压AHip测试气缸下降输出
ORLD
ANDLD
TIMX(550) 2211 E0_10  ; 短行程气缸报警延时, 4ST-1热压A下层Hip测试气缸下降位异常延时
LD TR0
LD T2211  ; 4ST-1热压A下层Hip测试气缸下降位异常延时
OR W405.11  ; 4ST-1热压A下层Hip测试气缸下降位异常
ANDLD
ANDNOT T0103  ; 复位按钮延时
OUT W405.11  ; 4ST-1热压A下层Hip测试气缸下降位异常
; rung 34
LD T0000  ; PLC上电延时5S
OUT TR0
LD H50.00  ; 4ST_1热压A上层有料记忆
ANDNOT T0184  ; 热压A上层有料感应延时
LDNOT H50.00  ; 4ST_1热压A上层有料记忆
AND T0184  ; 热压A上层有料感应延时
AND T0166  ; 出料夹爪上升位延时
AND T0156  ; 进料夹爪上升位延时
ORLD
ANDLD
TIMX(550) 2212 E0_10  ; 短行程气缸报警延时, 4ST-1热压A上层有料感应异常延时
LD TR0
LD T2212  ; 4ST-1热压A上层有料感应异常延时
OR W405.12  ; 4ST-1热压A上层有料感应异常
ANDLD
ANDNOT T0103  ; 复位按钮延时
OUT W405.12  ; 4ST-1热压A上层有料感应异常
; rung 35
LD T0000  ; PLC上电延时5S
OUT TR0
LD H50.01  ; 4ST_1热压A下层有料记忆
ANDNOT T0185  ; 热压A下层有料感应延时
LDNOT H50.01  ; 4ST_1热压A下层有料记忆
AND T0185  ; 热压A下层有料感应延时
AND T0166  ; 出料夹爪上升位延时
AND T0156  ; 进料夹爪上升位延时
ORLD
ANDLD
TIMX(550) 2213 E0_10  ; 短行程气缸报警延时, 4ST-1热压A下层有料感应异常延时
LD TR0
LD T2213  ; 4ST-1热压A下层有料感应异常延时
OR W405.13  ; 4ST-1热压A下层有料感应异常
ANDLD
ANDNOT T0103  ; 复位按钮延时
OUT W405.13  ; 4ST-1热压A下层有料感应异常

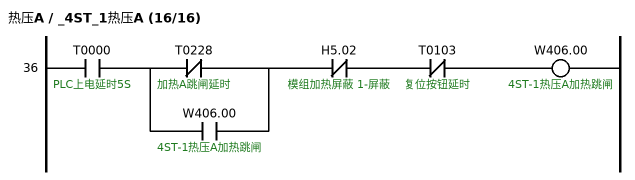
; rung 36
LD T0000  ; PLC上电延时5S
LDNOT T0228  ; 加热A跳闸延时
OR W406.00  ; 4ST-1热压A加热跳闸
ANDLD
ANDNOT H5.02  ; 模组加热屏蔽 1-屏蔽
ANDNOT T0103  ; 复位按钮延时
OUT W406.00  ; 4ST-1热压A加热跳闸

### Section 复位

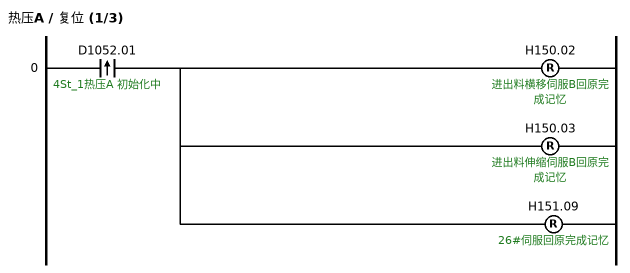
; rung 0
@LD D1052.01  ; 4St_1热压A 初始化中
RSET H150.02  ; 进出料横移伺服B回原完成记忆
RSET H150.03  ; 进出料伸缩伺服B回原完成记忆
RSET H151.09  ; 26#伺服回原完成记忆

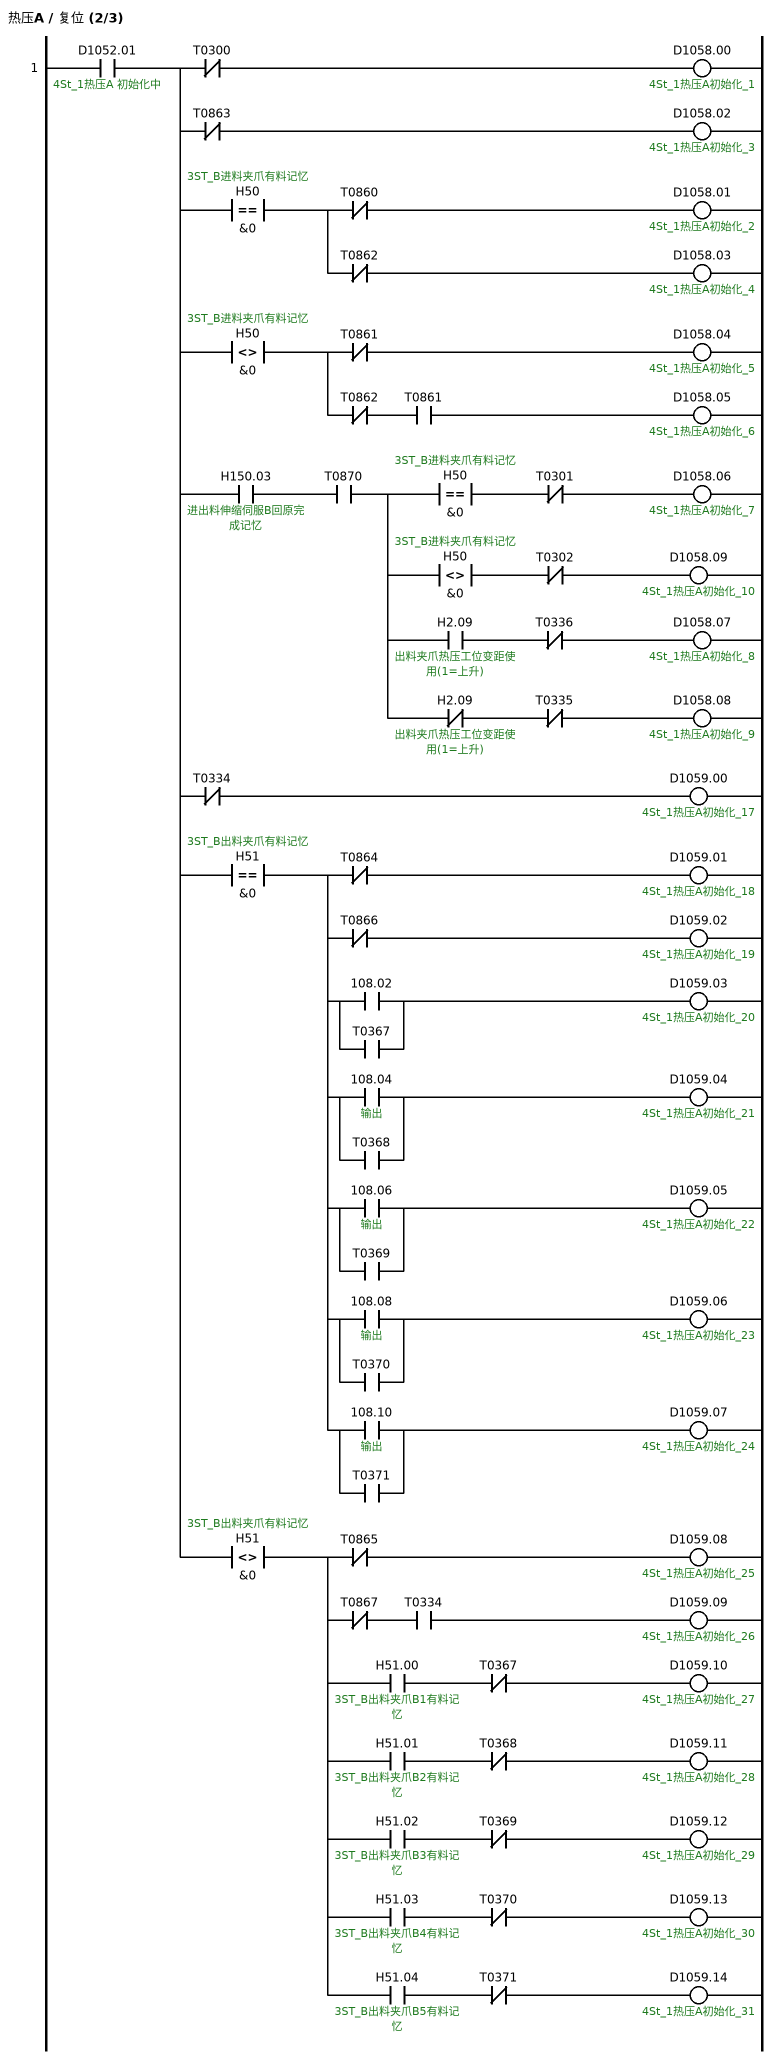
; rung 1
LD D1052.01  ; 4St_1热压A 初始化中
OUT TR0
ANDNOT T0300
OUT D1058.00  ; 4St_1热压A初始化_1
LD TR0
ANDNOT T0863
OUT D1058.02  ; 4St_1热压A初始化_3
LD TR0
AND=(300) H50 &0  ; 3ST_B进料夹爪有料记忆
OUT TR1
ANDNOT T0860
OUT D1058.01  ; 4St_1热压A初始化_2
LD TR1
ANDNOT T0862
OUT D1058.03  ; 4St_1热压A初始化_4
LD TR0
AND<>(305) H50 &0  ; 3ST_B进料夹爪有料记忆
OUT TR1
ANDNOT T0861
OUT D1058.04  ; 4St_1热压A初始化_5
LD TR1
ANDNOT T0862
AND T0861
OUT D1058.05  ; 4St_1热压A初始化_6
LD TR0
AND H150.03  ; 进出料伸缩伺服B回原完成记忆
AND T0870
OUT TR1
AND=(300) H50 &0  ; 3ST_B进料夹爪有料记忆
ANDNOT T0301
OUT D1058.06  ; 4St_1热压A初始化_7
LD TR1
AND<>(305) H50 &0  ; 3ST_B进料夹爪有料记忆
ANDNOT T0302
OUT D1058.09  ; 4St_1热压A初始化_10
LD TR1
AND H2.09  ; 出料夹爪热压工位变距使用(1=上升)
ANDNOT T0336
OUT D1058.07  ; 4St_1热压A初始化_8
LD TR1
ANDNOT H2.09  ; 出料夹爪热压工位变距使用(1=上升)
ANDNOT T0335
OUT D1058.08  ; 4St_1热压A初始化_9
LD TR0
ANDNOT T0334
OUT D1059.00  ; 4St_1热压A初始化_17
LD TR0
AND=(300) H51 &0  ; 3ST_B出料夹爪有料记忆
OUT TR1
ANDNOT T0864
OUT D1059.01  ; 4St_1热压A初始化_18
LD TR1
ANDNOT T0866
OUT D1059.02  ; 4St_1热压A初始化_19
LD TR1
LD 108.02
OR T0367
ANDLD
OUT D1059.03  ; 4St_1热压A初始化_20
LD TR1
LD 108.04  ; 输出
OR T0368
ANDLD
OUT D1059.04  ; 4St_1热压A初始化_21
LD TR1
LD 108.06  ; 输出
OR T0369
ANDLD
OUT D1059.05  ; 4St_1热压A初始化_22
LD TR1
LD 108.08  ; 输出
OR T0370
ANDLD
OUT D1059.06  ; 4St_1热压A初始化_23
LD TR1
LD 108.10  ; 输出
OR T0371
ANDLD
OUT D1059.07  ; 4St_1热压A初始化_24
LD TR0
AND<>(305) H51 &0  ; 3ST_B出料夹爪有料记忆
OUT TR0
ANDNOT T0865
OUT D1059.08  ; 4St_1热压A初始化_25
LD TR0
ANDNOT T0867
AND T0334
OUT D1059.09  ; 4St_1热压A初始化_26
LD TR0
AND H51.00  ; 3ST_B出料夹爪B1有料记忆
ANDNOT T0367
OUT D1059.10  ; 4St_1热压A初始化_27
LD TR0
AND H51.01  ; 3ST_B出料夹爪B2有料记忆
ANDNOT T0368
OUT D1059.11  ; 4St_1热压A初始化_28
LD TR0
AND H51.02  ; 3ST_B出料夹爪B3有料记忆
ANDNOT T0369
OUT D1059.12  ; 4St_1热压A初始化_29
LD TR0
AND H51.03  ; 3ST_B出料夹爪B4有料记忆
ANDNOT T0370
OUT D1059.13  ; 4St_1热压A初始化_30
LD TR0
AND H51.04  ; 3ST_B出料夹爪B5有料记忆
ANDNOT T0371
OUT D1059.14  ; 4St_1热压A初始化_31

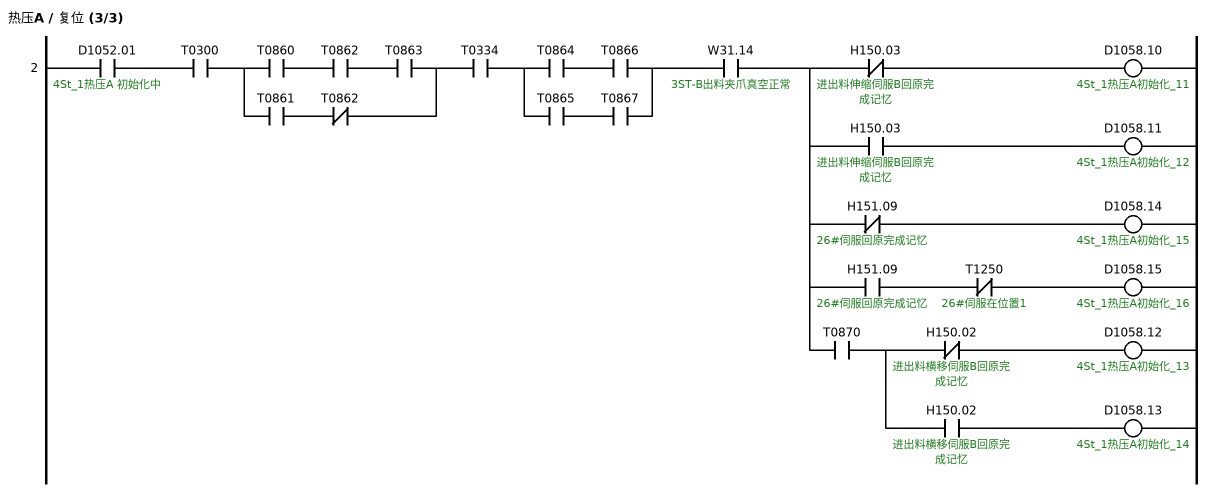
; rung 2
LD D1052.01  ; 4St_1热压A 初始化中
AND T0300
LD T0860
AND T0862
AND T0863
LD T0861
ANDNOT T0862
ORLD
ANDLD
AND T0334
LD T0864
AND T0866
LD T0865
AND T0867
ORLD
ANDLD
AND W31.14  ; 3ST-B出料夹爪真空正常
OUT TR0
ANDNOT H150.03  ; 进出料伸缩伺服B回原完成记忆
OUT D1058.10  ; 4St_1热压A初始化_11
LD TR0
AND H150.03  ; 进出料伸缩伺服B回原完成记忆
OUT D1058.11  ; 4St_1热压A初始化_12
LD TR0
ANDNOT H151.09  ; 26#伺服回原完成记忆
OUT D1058.14  ; 4St_1热压A初始化_15
LD TR0
AND H151.09  ; 26#伺服回原完成记忆
ANDNOT T1250  ; 26#伺服在位置1
OUT D1058.15  ; 4St_1热压A初始化_16
LD TR0
AND T0870
OUT TR0
ANDNOT H150.02  ; 进出料横移伺服B回原完成记忆
OUT D1058.12  ; 4St_1热压A初始化_13
LD TR0
AND H150.02  ; 进出料横移伺服B回原完成记忆
OUT D1058.13  ; 4St_1热压A初始化_14

### Section 输出

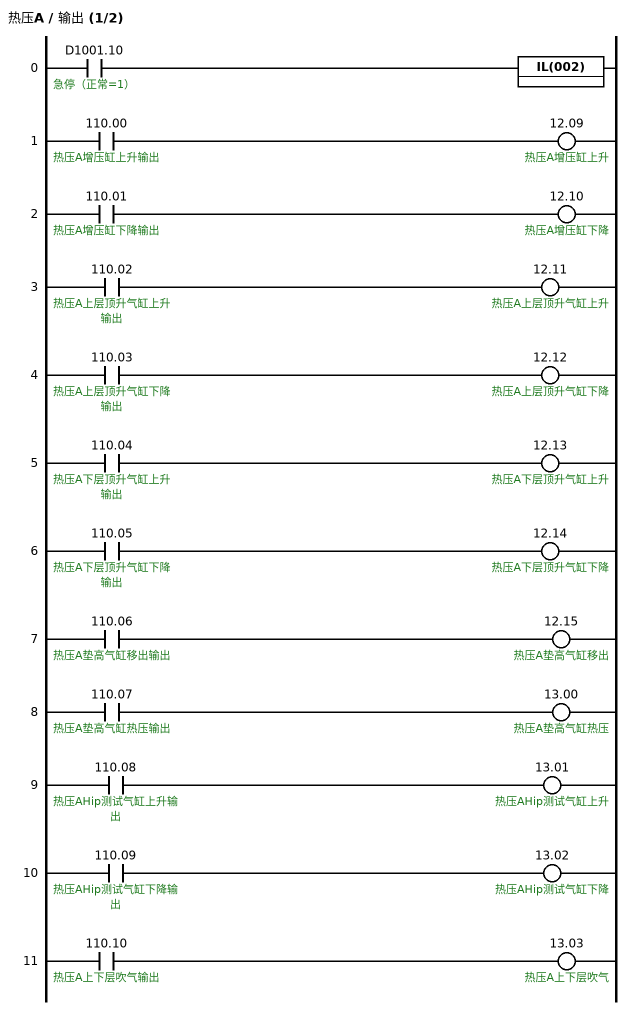
; rung 0
LD D1001.10  ; 急停（正常=1）
IL(002)
; rung 1
LD 110.00  ; 热压A增压缸上升输出
OUT 12.09  ; 热压A增压缸上升
; rung 2
LD 110.01  ; 热压A增压缸下降输出
OUT 12.10  ; 热压A增压缸下降
; rung 3
LD 110.02  ; 热压A上层顶升气缸上升输出
OUT 12.11  ; 热压A上层顶升气缸上升
; rung 4
LD 110.03  ; 热压A上层顶升气缸下降输出
OUT 12.12  ; 热压A上层顶升气缸下降
; rung 5
LD 110.04  ; 热压A下层顶升气缸上升输出
OUT 12.13  ; 热压A下层顶升气缸上升
; rung 6
LD 110.05  ; 热压A下层顶升气缸下降输出
OUT 12.14  ; 热压A下层顶升气缸下降
; rung 7
LD 110.06  ; 热压A垫高气缸移出输出
OUT 12.15  ; 热压A垫高气缸移出
; rung 8
LD 110.07  ; 热压A垫高气缸热压输出
OUT 13.00  ; 热压A垫高气缸热压
; rung 9
LD 110.08  ; 热压AHip测试气缸上升输出
OUT 13.01  ; 热压AHip测试气缸上升
; rung 10
LD 110.09  ; 热压AHip测试气缸下降输出
OUT 13.02  ; 热压AHip测试气缸下降
; rung 11
LD 110.10  ; 热压A上下层吹气输出
OUT 13.03  ; 热压A上下层吹气

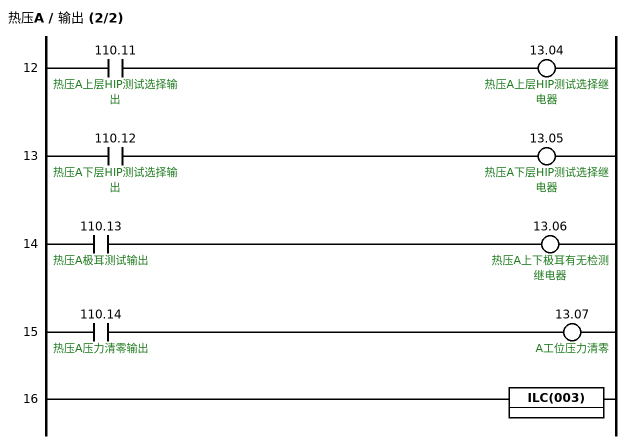
; rung 12
LD 110.11  ; 热压A上层HIP测试选择输出
OUT 13.04  ; 热压A上层HIP测试选择继电器
; rung 13
LD 110.12  ; 热压A下层HIP测试选择输出
OUT 13.05  ; 热压A下层HIP测试选择继电器
; rung 14
LD 110.13  ; 热压A极耳测试输出
OUT 13.06  ; 热压A上下极耳有无检测继电器
; rung 15
LD 110.14  ; 热压A压力清零输出
OUT 13.07  ; A工位压力清零
; rung 16
ILC(003)

### Section END
; rung 0
END(001)

## Program 热压B (cyclic task 5)
Local symbols
p_1s BOOL

### Section Main

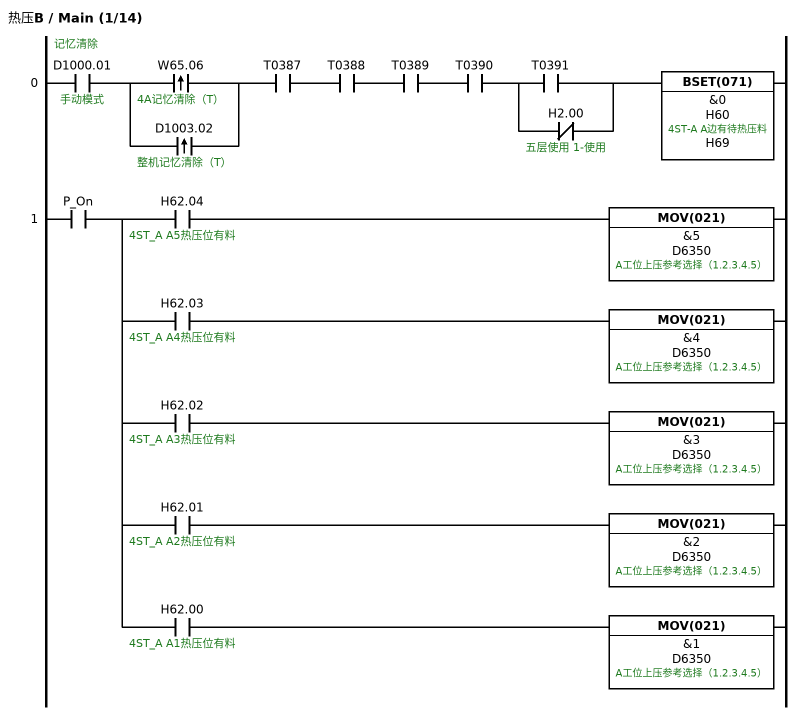
; rung 0: 记忆清除
LD D1000.01  ; 手动模式
@LD W65.06  ; 4A记忆清除（T）
@OR D1003.02  ; 整机记忆清除（T）
ANDLD
AND T0387
AND T0388
AND T0389
AND T0390
LD T0391
ORNOT H2.00  ; 五层使用 1-使用
ANDLD
BSET(071) &0 H60 H69  ; 4ST-A A边有待热压料
; rung 1
LD P_On
OUT TR0
AND H62.04  ; 4ST_A A5热压位有料
MOV(021) &5 D6350  ; A工位上压参考选择（1.2.3.4.5）
LD TR0
AND H62.03  ; 4ST_A A4热压位有料
MOV(021) &4 D6350  ; A工位上压参考选择（1.2.3.4.5）
LD TR0
AND H62.02  ; 4ST_A A3热压位有料
MOV(021) &3 D6350  ; A工位上压参考选择（1.2.3.4.5）
LD TR0
AND H62.01  ; 4ST_A A2热压位有料
MOV(021) &2 D6350  ; A工位上压参考选择（1.2.3.4.5）
LD TR0
AND H62.00  ; 4ST_A A1热压位有料
MOV(021) &1 D6350  ; A工位上压参考选择（1.2.3.4.5）

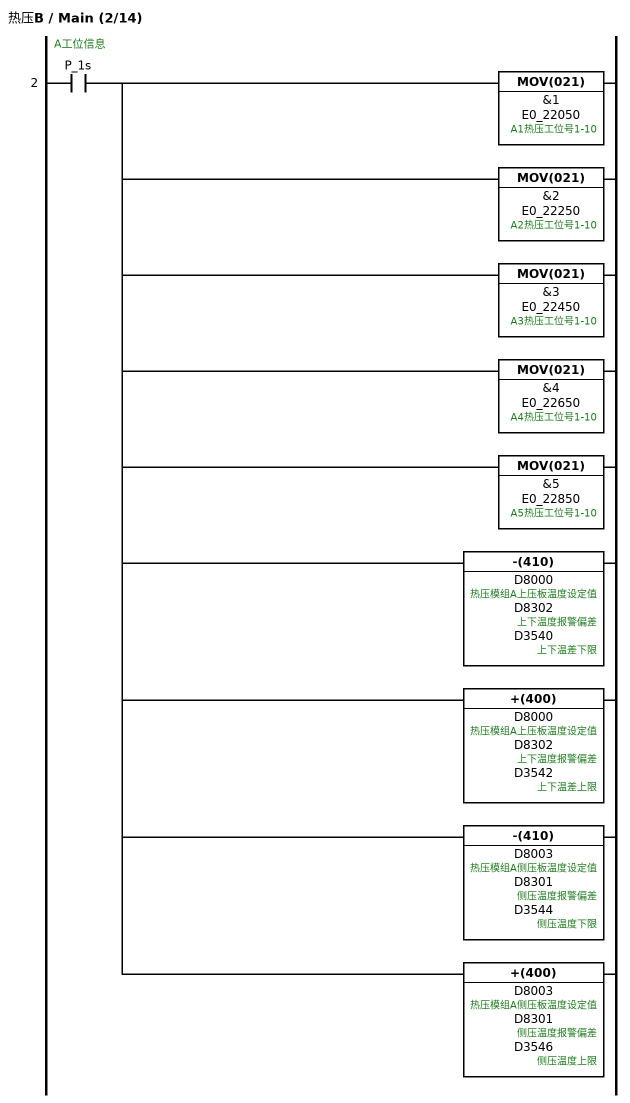
; rung 2: A工位信息
LD P_1s
MOV(021) &1 E0_22050  ; A1热压工位号1-10
MOV(021) &2 E0_22250  ; A2热压工位号1-10
MOV(021) &3 E0_22450  ; A3热压工位号1-10
MOV(021) &4 E0_22650  ; A4热压工位号1-10
MOV(021) &5 E0_22850  ; A5热压工位号1-10
-(410) D8000 D8302 D3540  ; 热压模组A上压板温度设定值, 上下温度报警偏差, 上下温差下限
+(400) D8000 D8302 D3542  ; 热压模组A上压板温度设定值, 上下温度报警偏差, 上下温差上限
-(410) D8003 D8301 D3544  ; 热压模组A侧压板温度设定值, 侧压温度报警偏差, 侧压温度下限
+(400) D8003 D8301 D3546  ; 热压模组A侧压板温度设定值, 侧压温度报警偏差, 侧压温度上限

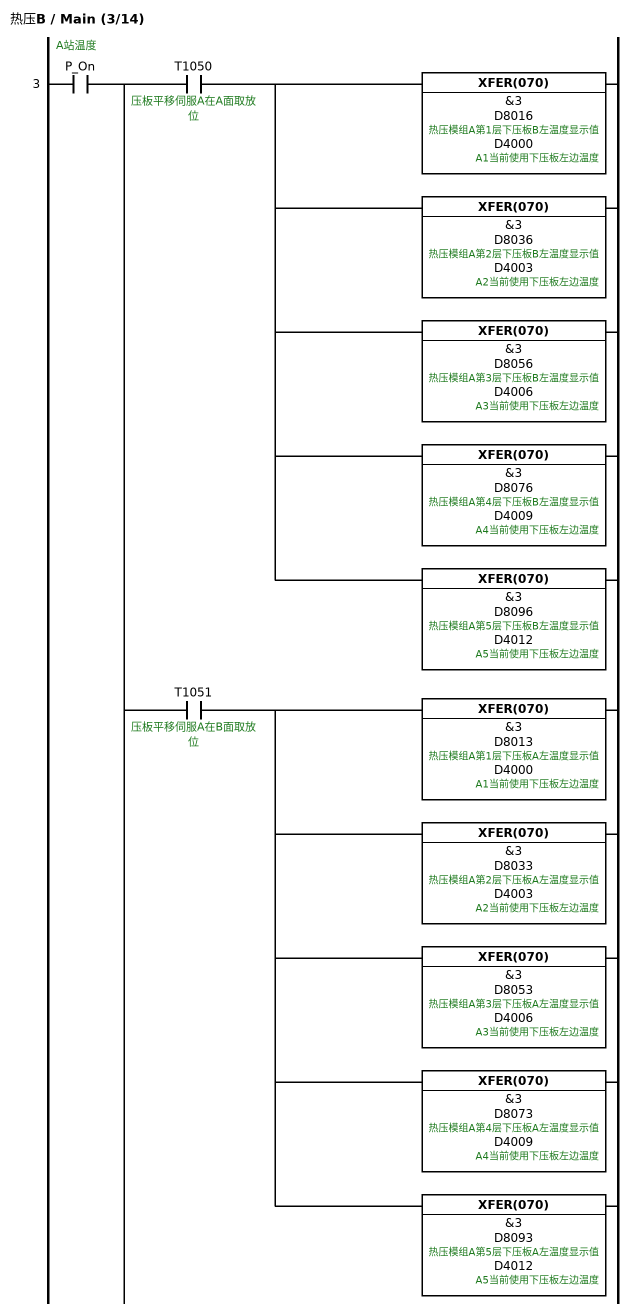

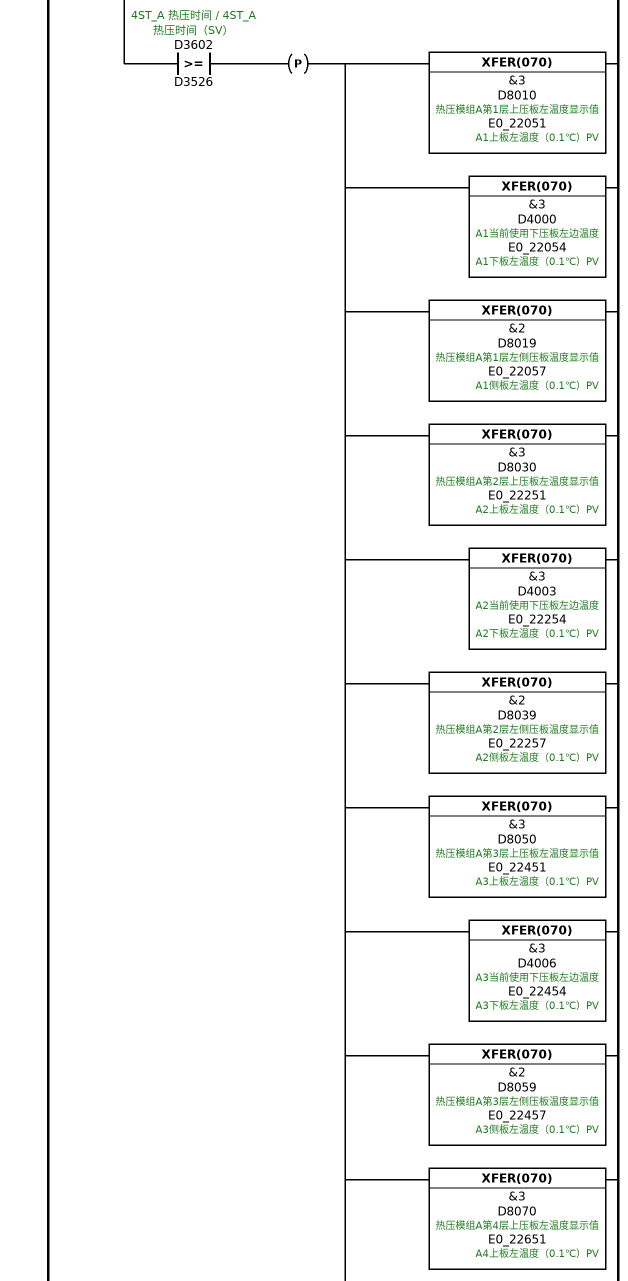

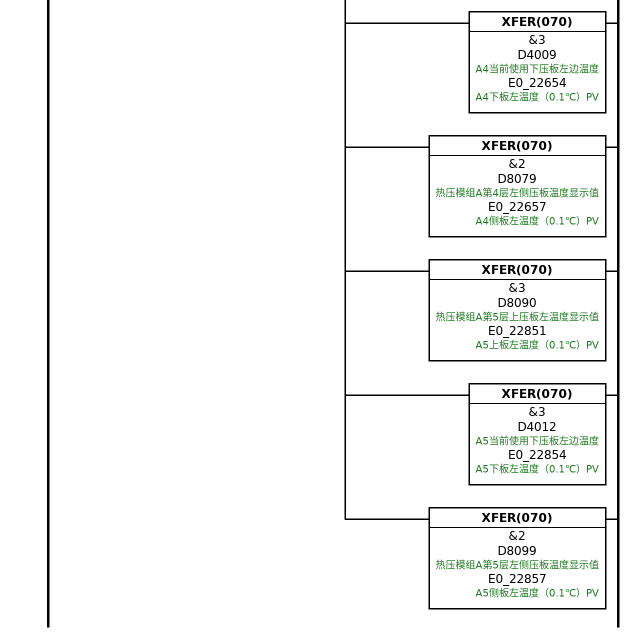
; rung 3: A站温度
LD P_On
OUT TR0
AND T1050  ; 压板平移伺服A在A面取放位
XFER(070) &3 D8016 D4000  ; 热压模组A第1层下压板B左温度显示值, A1当前使用下压板左边温度
XFER(070) &3 D8036 D4003  ; 热压模组A第2层下压板B左温度显示值, A2当前使用下压板左边温度
XFER(070) &3 D8056 D4006  ; 热压模组A第3层下压板B左温度显示值, A3当前使用下压板左边温度
XFER(070) &3 D8076 D4009  ; 热压模组A第4层下压板B左温度显示值, A4当前使用下压板左边温度
XFER(070) &3 D8096 D4012  ; 热压模组A第5层下压板B左温度显示值, A5当前使用下压板左边温度
LD TR0
AND T1051  ; 压板平移伺服A在B面取放位
XFER(070) &3 D8013 D4000  ; 热压模组A第1层下压板A左温度显示值, A1当前使用下压板左边温度
XFER(070) &3 D8033 D4003  ; 热压模组A第2层下压板A左温度显示值, A2当前使用下压板左边温度
XFER(070) &3 D8053 D4006  ; 热压模组A第3层下压板A左温度显示值, A3当前使用下压板左边温度
XFER(070) &3 D8073 D4009  ; 热压模组A第4层下压板A左温度显示值, A4当前使用下压板左边温度
XFER(070) &3 D8093 D4012  ; 热压模组A第5层下压板A左温度显示值, A5当前使用下压板左边温度
LD TR0
AND>=(325) D3602 D3526  ; 4ST_A 热压时间, 4ST_A 热压时间（SV）
UP(521)
XFER(070) &3 D8010 E0_22051  ; 热压模组A第1层上压板左温度显示值, A1上板左温度（0.1℃）PV
XFER(070) &3 D4000 E0_22054  ; A1当前使用下压板左边温度, A1下板左温度（0.1℃）PV
XFER(070) &2 D8019 E0_22057  ; 热压模组A第1层左侧压板温度显示值, A1侧板左温度（0.1℃）PV
XFER(070) &3 D8030 E0_22251  ; 热压模组A第2层上压板左温度显示值, A2上板左温度（0.1℃）PV
XFER(070) &3 D4003 E0_22254  ; A2当前使用下压板左边温度, A2下板左温度（0.1℃）PV
XFER(070) &2 D8039 E0_22257  ; 热压模组A第2层左侧压板温度显示值, A2侧板左温度（0.1℃）PV
XFER(070) &3 D8050 E0_22451  ; 热压模组A第3层上压板左温度显示值, A3上板左温度（0.1℃）PV
XFER(070) &3 D4006 E0_22454  ; A3当前使用下压板左边温度, A3下板左温度（0.1℃）PV
XFER(070) &2 D8059 E0_22457  ; 热压模组A第3层左侧压板温度显示值, A3侧板左温度（0.1℃）PV
XFER(070) &3 D8070 E0_22651  ; 热压模组A第4层上压板左温度显示值, A4上板左温度（0.1℃）PV
XFER(070) &3 D4009 E0_22654  ; A4当前使用下压板左边温度, A4下板左温度（0.1℃）PV
XFER(070) &2 D8079 E0_22657  ; 热压模组A第4层左侧压板温度显示值, A4侧板左温度（0.1℃）PV
XFER(070) &3 D8090 E0_22851  ; 热压模组A第5层上压板左温度显示值, A5上板左温度（0.1℃）PV
XFER(070) &3 D4012 E0_22854  ; A5当前使用下压板左边温度, A5下板左温度（0.1℃）PV
XFER(070) &2 D8099 E0_22857  ; 热压模组A第5层左侧压板温度显示值, A5侧板左温度（0.1℃）PV

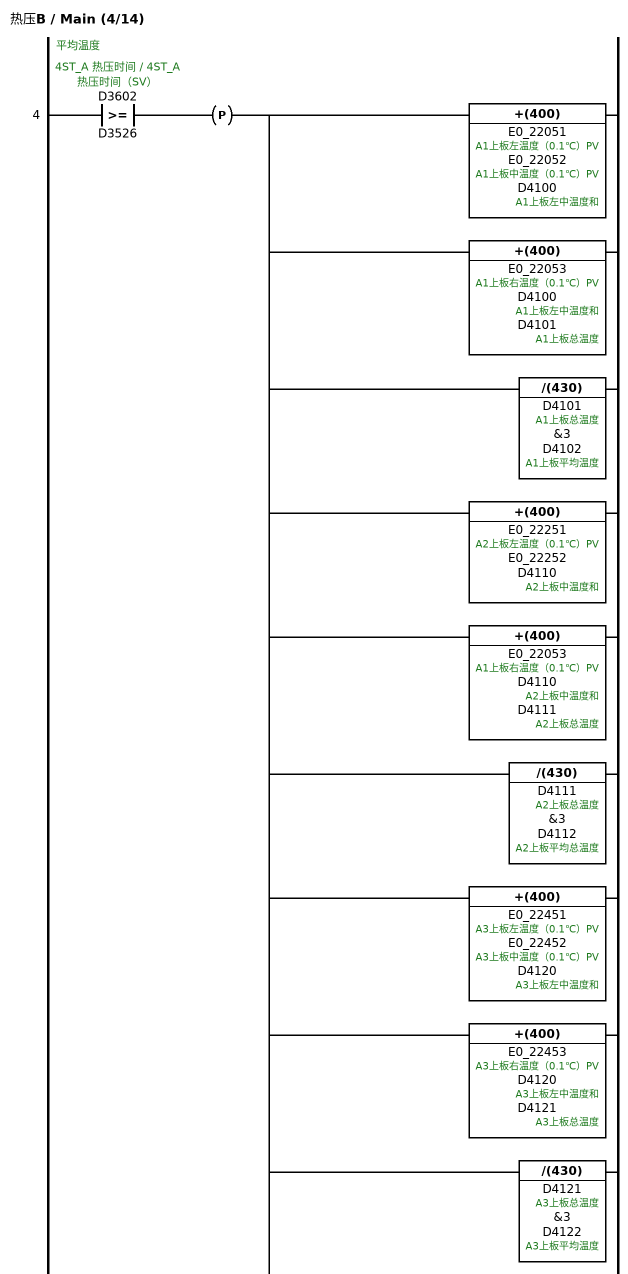

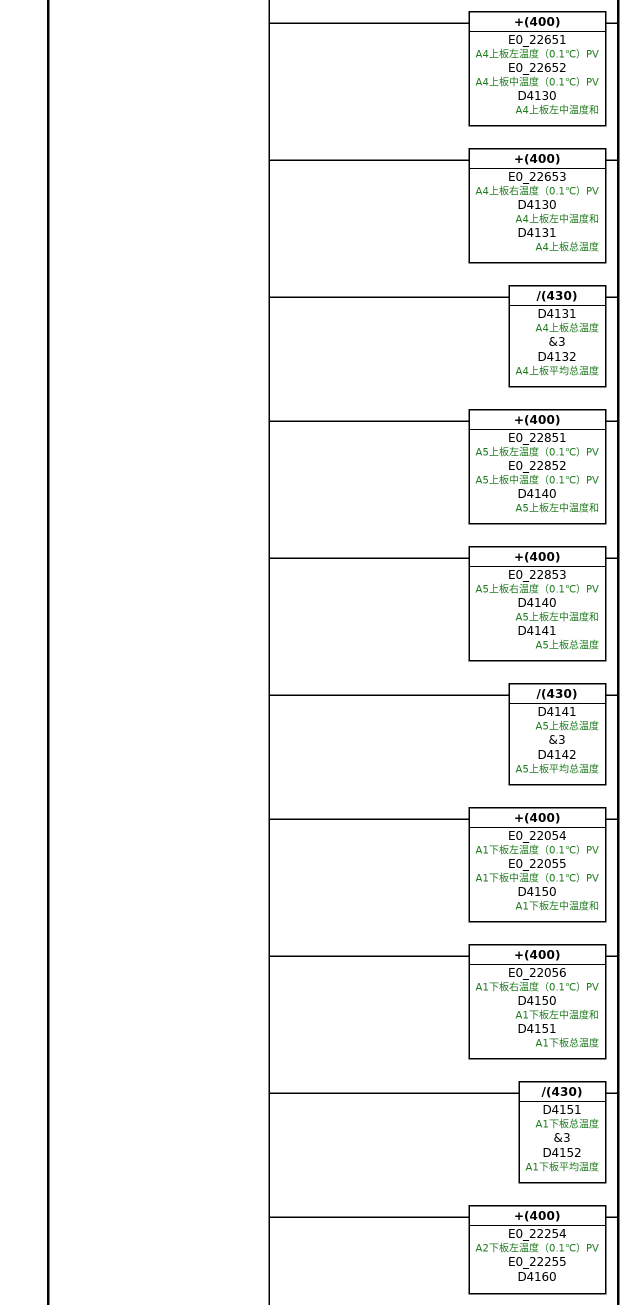

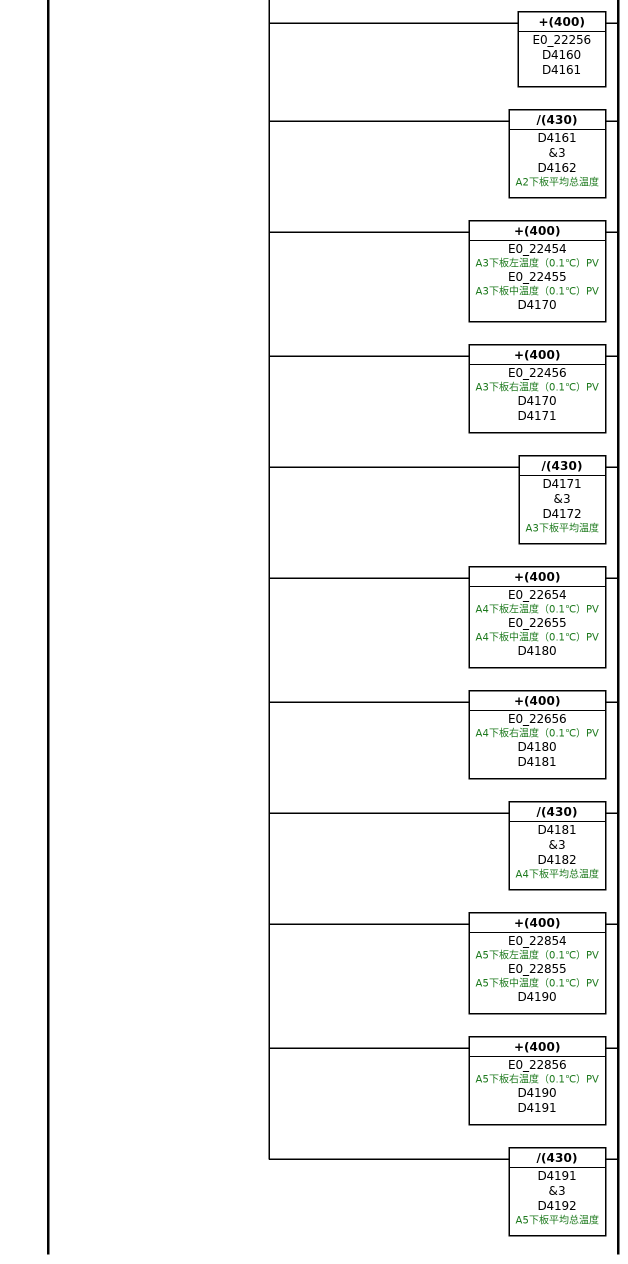
; rung 4: 平均温度
LD>=(325) D3602 D3526  ; 4ST_A 热压时间, 4ST_A 热压时间（SV）
UP(521)
+(400) E0_22051 E0_22052 D4100  ; A1上板左温度（0.1℃）PV, A1上板中温度（0.1℃）PV, A1上板左中温度和
+(400) E0_22053 D4100 D4101  ; A1上板右温度（0.1℃）PV, A1上板左中温度和, A1上板总温度
/(430) D4101 &3 D4102  ; A1上板总温度, A1上板平均温度
+(400) E0_22251 E0_22252 D4110  ; A2上板左温度（0.1℃）PV, A2上板中温度和
+(400) E0_22053 D4110 D4111  ; A1上板右温度（0.1℃）PV, A2上板中温度和, A2上板总温度
/(430) D4111 &3 D4112  ; A2上板总温度, A2上板平均总温度
+(400) E0_22451 E0_22452 D4120  ; A3上板左温度（0.1℃）PV, A3上板中温度（0.1℃）PV, A3上板左中温度和
+(400) E0_22453 D4120 D4121  ; A3上板右温度（0.1℃）PV, A3上板左中温度和, A3上板总温度
/(430) D4121 &3 D4122  ; A3上板总温度, A3上板平均温度
+(400) E0_22651 E0_22652 D4130  ; A4上板左温度（0.1℃）PV, A4上板中温度（0.1℃）PV, A4上板左中温度和
+(400) E0_22653 D4130 D4131  ; A4上板右温度（0.1℃）PV, A4上板左中温度和, A4上板总温度
/(430) D4131 &3 D4132  ; A4上板总温度, A4上板平均总温度
+(400) E0_22851 E0_22852 D4140  ; A5上板左温度（0.1℃）PV, A5上板中温度（0.1℃）PV, A5上板左中温度和
+(400) E0_22853 D4140 D4141  ; A5上板右温度（0.1℃）PV, A5上板左中温度和, A5上板总温度
/(430) D4141 &3 D4142  ; A5上板总温度, A5上板平均总温度
+(400) E0_22054 E0_22055 D4150  ; A1下板左温度（0.1℃）PV, A1下板中温度（0.1℃）PV, A1下板左中温度和
+(400) E0_22056 D4150 D4151  ; A1下板右温度（0.1℃）PV, A1下板左中温度和, A1下板总温度
/(430) D4151 &3 D4152  ; A1下板总温度, A1下板平均温度
+(400) E0_22254 E0_22255 D4160  ; A2下板左温度（0.1℃）PV
+(400) E0_22256 D4160 D4161
/(430) D4161 &3 D4162  ; A2下板平均总温度
+(400) E0_22454 E0_22455 D4170  ; A3下板左温度（0.1℃）PV, A3下板中温度（0.1℃）PV
+(400) E0_22456 D4170 D4171  ; A3下板右温度（0.1℃）PV
/(430) D4171 &3 D4172  ; A3下板平均温度
+(400) E0_22654 E0_22655 D4180  ; A4下板左温度（0.1℃）PV, A4下板中温度（0.1℃）PV
+(400) E0_22656 D4180 D4181  ; A4下板右温度（0.1℃）PV
/(430) D4181 &3 D4182  ; A4下板平均总温度
+(400) E0_22854 E0_22855 D4190  ; A5下板左温度（0.1℃）PV, A5下板中温度（0.1℃）PV
+(400) E0_22856 D4190 D4191  ; A5下板右温度（0.1℃）PV
/(430) D4191 &3 D4192  ; A5下板平均总温度

